        (* ***** Single Read SpecialFixcode ***** *)
        IF Head1.SaveRead AND NOT I_b_Head1SingleEnhanced AND I_b_Head1SpecialFixcode THEN
            Head_1_OutData[0] := 16#0A;
            Head_1_OutData[1] := 16#02;
            
            Head1.SglCommandActive := TRUE;
            Head1.EnhCommandActive := FALSE;
            Head1.Execute := TRUE;
            state_cmd1 := 1;
        END_IF;
        
        (* ***** Enhanced Read Words ***** *)
        IF Head1.SaveRead AND NOT I_b_Head1DataFixcode AND I_b_Head1SingleEnhanced AND NOT I_b_Head1SpecialFixcode THEN
            Head_1_OutData[0] := 16#19;
            Head_1_OutData[1] := WORD_TO_BYTE((INT_TO_WORD(SHL(I_i_Head1WordNum,  4)) OR 16#2));
            Head_1_OutData[2] := WORD_TO_BYTE(SHR(I_w_Head1WordAddress AND 16#FF00, 8));
            Head_1_OutData[3] := WORD_TO_BYTE(I_w_Head1WordAddress);
            
            Head1.EnhCommandActive := TRUE;
            Head1.Execute := TRUE;
            state_cmd1 := 1;
        END_IF;
        
        (* ***** Enhanced Read Fixcode ***** *)
        IF Head1.SaveRead AND I_b_Head1DataFixcode AND I_b_Head1SingleEnhanced AND NOT I_b_Head1SpecialFixcode THEN
            Head_1_OutData[0] := 16#1D;
            Head_1_OutData[1] := 16#02;
            
            Head1.EnhCommandActive := TRUE;
            Head1.Execute := TRUE;
            state_cmd1 := 1;
        END_IF;
        
        (* ***** Enhanced Read SpecialFixcode ***** *)
        IF Head1.SaveRead AND I_b_Head1SingleEnhanced AND I_b_Head1SpecialFixcode THEN
            Head_1_OutData[0] := 16#71;
            Head_1_OutData[1] := 16#02;
            
            Head1.EnhCommandActive := TRUE;
            Head1.Execute := TRUE;
            state_cmd1 := 1;
        END_IF;
        
        (* ***** Single Write Words ***** *)
        IF Head1.SaveWrite AND NOT I_b_Head1DataFixcode AND NOT I_b_Head1SingleEnhanced AND NOT I_b_Head1SpecialFixcode THEN
            Head_1_OutData[0] := 16#40;
            Head_1_OutData[1] := WORD_TO_BYTE((INT_TO_WORD(SHL(I_i_Head1WordNum, 4)) OR 16#2));
            Head_1_OutData[2] := WORD_TO_BYTE(SHR( I_w_Head1WordAddress AND 16#FF00,  8));
            Head_1_OutData[3] := WORD_TO_BYTE(I_w_Head1WordAddress);
            //Copy Write Data field to Out Data beginning at element [4]
            MEMCPY(srcAddr:=ADR(Head1Data.WriteData[0]) , destAddr:=ADR(Head_1_OutData[4]) , n:=SIZEOF(Head1Data.WriteData) );
			
            Head1.SglCommandActive := TRUE;
            Head1.EnhCommandActive := FALSE;
            Head1.Execute := TRUE;
            state_cmd1 := 1;
        END_IF;
        
        (* ***** Enhanced Write Words ***** *)
        IF Head1.SaveWrite AND NOT I_b_Head1DataFixcode AND I_b_Head1SingleEnhanced AND NOT I_b_Head1SpecialFixcode THEN
            Head_1_OutData[0] := 16#1A;
            Head_1_OutData[1] := WORD_TO_BYTE((INT_TO_WORD(SHL(I_i_Head1WordNum, 4)) OR 16#2));
            Head_1_OutData[2] := WORD_TO_BYTE(SHR( I_w_Head1WordAddress AND 16#FF00, 8));
            Head_1_OutData[3] := WORD_TO_BYTE(I_w_Head1WordAddress);
            //Copy Write Data field to Out Data beginning at element [4]		 
			MEMCPY(srcAddr:= ADR(Head1Data.WriteData[0]) , destAddr:=ADR(Head_1_OutData[4]) , n:=SIZEOF(Head1Data.WriteData) );		 
	 
            Head1.EnhCommandActive := TRUE;
            Head1.Execute := TRUE;
            state_cmd1 := 1;
        END_IF;
        
        (* ***** Single Write Fixcode ***** *) (* - default for IPC11, FixType = 11 & FixLen = 5 *)
        IF Head1.SaveWrite AND I_b_Head1DataFixcode AND NOT I_b_Head1SingleEnhanced AND NOT I_b_Head1SpecialFixcode THEN
            Head_1_OutData[0] := 16#1F;
            Head_1_OutData[1] := WORD_TO_BYTE((INT_TO_WORD(SHL(16#5,  4)) OR 16#2));
            Head_1_OutData[2] := 16#31; (* ASCII 11 = 0x3131, overwrite fixcode *)
            Head_1_OutData[3] := 16#31;
            //Copy Write Data field to Out Data beginning at element [4]
           MEMCPY(srcAddr:= ADR(Head1Data.WriteData[0]) , destAddr:=ADR(Head_1_OutData[4]) , n:=SIZEOF(Head1Data.WriteData) );
            	 
            Head1.SglCommandActive := TRUE;
            Head1.EnhCommandActive := FALSE;
            Head1.Execute := TRUE;
            state_cmd1 := 1;
        END_IF;
        
        (* ***** Single Write SpecialFixcode ***** *)
        IF Head1.SaveWrite AND NOT I_b_Head1SingleEnhanced AND I_b_Head1SpecialFixcode THEN
            Head_1_OutData[0] := 16#0D;
            Head_1_OutData[1] := WORD_TO_BYTE((INT_TO_WORD(SHL(I_i_Head1WordNum, 4)) OR 16#2));
            Head_1_OutData[2] := 16#0; (* reserved *)
            Head_1_OutData[3] := 16#0; (* reserved *)
            //Copy Write Data field to Out Data beginning at element [4]
            MEMCPY(srcAddr:= ADR(Head1Data.WriteData[0]) , destAddr:=ADR(Head_1_OutData[4]) , n:=SIZEOF(Head1Data.WriteData ));
		 
            Head1.SglCommandActive := TRUE;
            Head1.EnhCommandActive := FALSE;
            Head1.Execute := TRUE;
            state_cmd1 := 1;
        END_IF;
        
        (* ***** Special Command ***** *)
        IF Head1.SaveSpecialCommand AND NOT I_b_Head1SpecialFixcode THEN
        (* Copy SpecialCommand-Array into Output-Array *)
            //Copy the whole SpecialCommand data field to the Output Data
			 MEMCPY(srcAddr:=ADR(Head1Data.SpecialCommand[0]) , destAddr:=ADR(Head_1_OutData[0]) , n:=SIZEOF(Head1Data.SpecialCommand) );		 
			
            Head1.SglCommandActive := TRUE;
            Head1.EnhCommandActive := FALSE;
            Head1.Execute := TRUE;
            state_cmd1 := 1;
        END_IF;
    END_IF;
    
(* ***** Handle communication and analysis for channel 1 ***** *)
    CASE state_cmd1 OF
            
        0:  (* ***** Idle state ***** *)
//        IF NOT I_b_Head1SingleEnhanced
//			AND NOT	I_b_Head1DataFixcode
//			AND NOT	I_b_Head1SpecialFixcode
//			AND NOT	I_b_Head1SpecialCommand
//			AND NOT	I_b_Head1Read
//			AND NOT	I_b_Head1Write
//			AND NOT	I_b_Head1Quit
//			THEN
			O_b_Head1Done := FALSE;
			//O_b_Head1NoDataCarrier := FALSE;
//		END_IF

        1:  (* ***** Execution ***** *)
            IF Head1.Execute AND NOT Head1.TransfToHead THEN
                
                Head1.Busy := TRUE;
                O_b_Head1Busy := TRUE;
                Head1.Done := FALSE;
                O_b_Head1Done := FALSE;
                Head1.Error := FALSE;
                O_b_Head1Error := FALSE;
                Head1.SendOK := FALSE;
                Head1.ReceiveOK := FALSE;
                Head1.NoDataCarrier := FALSE;
                O_b_Head1NoDataCarrier := FALSE;
                Head1.NewData := FALSE;
                Head1.TimeoutActive := TRUE;
                Head1.TimeoutOccurred := FALSE;
                Head1.TransfToHead := TRUE;
                Head1.SaveRead := FALSE;
                Head1.SaveWrite := FALSE;
                Head1.SaveQuit := FALSE;
                Head1.SaveSpecialCommand := FALSE;
                
                (* Invert togglebit => new telegram is available *)
                IF Memory.Togglebit <> 1 THEN
                    Head_1_OutData[1] := Head_1_OutData[1] OR 16#1;
                ELSE
                    Head_1_OutData[1] := Head_1_OutData[1] AND 16#FE;
                END_IF;
                
               		HwOut:= Head_1_OutData ; (* Write on BUS *)
               
                 
                    state_cmd1 := state_cmd1 + 1; (* Go to next state *)
                
            END_IF;
            
            
        2:(* ***** Analyze InData ***** *)
        (* Receive Telegram *)
            IF Head1.NewData THEN
                
                Head1.NewData := FALSE;
                (* Transfer status & reply counter to output *)
                O_B_Head1Status := Head_1_InData[2];
                O_B_Head1ReplyCounter := Head_1_InData[3];
                
                (* Analyze status *)
                IF Head_1_InData[2] = 16#FF THEN
                    Head1.SendOK := TRUE;
                    Head1.TransfToHead := FALSE;
                ELSE
                    Head1.Execute := FALSE;
                    Head1.ReceiveOK := TRUE;
                    Head1.SglCommandActive := FALSE;
                    Head1.TimeoutActive := FALSE;
                    Head1.Busy := FALSE;
                    O_b_Head1Busy := FALSE;
                    Head1.Done := TRUE;
                    O_b_Head1Done := TRUE;
                    state_cmd1 := 0; (* Go to idle state *)
                END_IF;
                
                IF Head_1_InData[2] = 16#0 THEN
                    Head1.NoDataCarrier := FALSE;
                    O_b_Head1NoDataCarrier := FALSE;
                    Head1.Error := FALSE;      //new in 3.0
                    O_b_Head1Error := FALSE;       //new in 3.0
                END_IF;
                
                IF Head_1_InData[2] = 16#5 THEN
                    Head1.NoDataCarrier := TRUE;
                    O_b_Head1NoDataCarrier := TRUE;
                    Head1.Error := FALSE;      //new in 3.0
                    O_b_Head1Error := FALSE;       //new in 3.0
                END_IF;
                
                (* Error states *)
                IF Head_1_InData[2] = 16#4
                    OR Head_1_InData[2] = 16#6
                    OR Head_1_InData[2] = 16#7
                    OR Head_1_InData[2] = 16#9
                    OR Head_1_InData[2] = 16#A
                    OR Head_1_InData[2] = 16#E THEN
                    Head1.Error := TRUE;
                    O_b_Head1Error := TRUE;
                END_IF;
                
                (* Different output behaviour during active enhanced command *)
                IF Head1.EnhCommandActive THEN
                    state_cmd1 := 2; (* Receive new telegram *)
                    Head1.Busy := TRUE;
                    O_b_Head1Busy := TRUE;
                    IF Head_1_InData[2] = 16#0 THEN
                        Head1.Done := TRUE;
                        O_b_Head1Done := TRUE;
                    ELSE
                        Head1.Done := FALSE;
                        O_b_Head1Done := FALSE;
                    END_IF;
                END_IF;
            END_IF;
    END_CASE;
	
	
END_IF;

(* ***** Watchdog ***** *)
//Watchdog1(IN := Head1.TimeoutActive,PT := I_T_Timeout);

IF (Watchdog1.Q AND temp) THEN
    Head1.TimeoutActive := FALSE;
    Head1.TimeoutOccurred := TRUE;
    Head1.SendOK := FALSE;
    Head1.ReceiveOK := FALSE;
    Head1.SglCommandActive := FALSE;
    Head1.EnhCommandActive := FALSE;
    Head1.Execute := FALSE;
    Head1.TransfToHead := FALSE;
    Head1.Error := TRUE;
    O_b_Head1Error := TRUE;
    Head1.Busy := FALSE;
    O_b_Head1Busy := FALSE;
    Head1.Done := TRUE;
    O_b_Head1Done := TRUE;
END_IF

END_FUNCTION_BLOCK

// ---- POUs/Programs/OP10/OP10_MAIN.TcPOU
PROGRAM OP10_MAIN
VAR

	OP10A_ROBO_MANUL_TRG: R_TRIG;
	OP10A_ROBO_AUTO_TRG	: R_TRIG;
	Bowl_A_ON_Timer		: TON;
	Bowl_A_OFF_Timer	: TON;
	Bowl_B_ON_Timer		: TON;
	Bowl_B_OFF_Timer	: TON;
	OP10A_ROBO_ERR		: TON;
	OP10B_ROBO_ERR		: TON;
	SRV_HOME			: BOOL;	
	OP10_ROBO			: INT;
	OP10A_ROBO_MANUAL	: INT;
	OP10A_ROBO_AUTO		: INT;
	// TEMP
	TEMP_40				: BOOL;

	

	
	OP10B_ROBO_MANUL_TRG: R_TRIG;
	OP10B_ROBO_AUTO_TRG: R_TRIG;
	OP10B_ROBO_MANUAL: INT;
	OP10B_ROBO_AUTO: INT;
END_VAR

VAR PERSISTENT
	OP10A_ROBO_ERR_TIME	: TIME;
	OP10B_ROBO_ERR_TIME	: TIME;
END_VAR

OP10_MANUAL();
OP10_SERVO();
OP10_HOMING();
OP10A_AUTO();
OP10B_AUTO();
//OP10_AUTO();
Bowl_Control();
OP10A_Camera_FB();
OP10B_Camera_FB();
OP10A_OP10B_DRUM_FEEDER();
OP10B_Conveyor_Prog();
OP10A_Conveyor_Prog();
//OP10_Body_Camera_Seq();
Body_Singulation_Seq();

OP10A_MODE_BLOCK(
	ModeWord:= OP10A_MODE_WORD, 
	HomeConditionOK:= OP10A_ALL_HOME,//OP10A_ALL_HOME, 
	OperationEnable:= OperationEnable, 
	StartPB:= OP10A_STRT_PB, 
	SafetyAndNOError:= NOT OP10A_ERR,//(NOT OP10A_ERR), 
	ModeAck:= 1, 
	HomingINProgress:= , 
	TempHomeOK:=  , 
	ResetPB:= Servo_Reset, 
	AutoSelected=> OP10A_AUTO_SELECTED, 
	ManualSelected=> OP10A_MANUAL_SELECTED, 
	StepSelected=> OP10A_STEP_SELECTED, 
	ModeSelAck_Indication=> , 
	StatusDisplay=> , 
	AutoRunning:=OP10A_AUTO_RUNNING, 
	StepRunning:=OP10A_STEP_RUNNING , 
	StartEnable:=OP10A_START_ENABLE , 
	MachineStop:=OP10A_MACHINE_STOP );
	
	
	OP10A_ROBO_MANUL_TRG(CLK:=OP10A_MANUAL_SELECTED , Q=> );
	OP10A_ROBO_AUTO_TRG(CLK:=NOT OP10A_MANUAL_SELECTED , Q=> );
	
IF OP10A_ROBO_MANUL_TRG.Q THEN
	OP10A_ROBO_MANUAL	:= 1;
END_IF

IF OP10A_ROBO_AUTO_TRG.Q THEN
	OP10A_ROBO_AUTO		:= 1;
END_IF


CASE OP10A_ROBO_MANUAL OF 
	1: OP10A_ROBO_PRGM_RST				:= TRUE;
		OP10A_ROBO_MANUAL				:= 5;
		
	5: IF (OP10A_ROBO_PRGM_RST =TRUE) AND (NOT OP10A_Program_Execute) THEN
		OP10A_ROBO_PRGM_RST				:= FALSE;
		O10A_ROB_MAN_AUTO_MODE_Q709_2	:= FALSE;
		OP10A_ROBO_MANUAL				:= 10;
		END_IF
END_CASE

CASE OP10A_ROBO_AUTO OF 
	1: OP10A_ROBO_PRGM_RST				:= TRUE;
		OP10A_ROBO_AUTO					:= 5;

	5: IF (OP10A_ROBO_PRGM_RST =TRUE) AND (NOT OP10A_Program_Execute) THEN
		OP10A_ROBO_PRGM_RST				:= FALSE;
		O10A_ROB_MAN_AUTO_MODE_Q709_2	:= TRUE;
		OP10A_ROBO_AUTO					:= 10;
		END_IF
END_CASE


OP10A_ROBO_ERR(IN:=	NOT(OP10A_Auto_Operation_Enable AND OP10A_Mirror_Auto_enable AND OP10A_Servo_ON_OFF_Status) , PT:=OP10A_ROBO_ERR_TIME, Q=> , ET=> );
			
IF (OP10A_AUTO_SELECTED AND NOT OP10A_ROBO_PRGM_RST AND OP10A_ROBO_ERR.Q) OR OP10A_H_Error OR OP10A_L_Error OR 
		OP10_SRV_FRST_PCKBDY_CNT.Axis_Error OR OP10_SRV_SCND_PCKBDY_CNT.Axis_Error OR(OP10A_CYLINDER_ERR<>0) OR 
			(OP10A_SRV_LH_BDYANG_CNT.Axis_Error AND NOT OP10A_BDY1_PCK_BYPAS) OR (OP10A_SRV_RH_BDYANG_CNT.Axis_Error AND 
				NOT OP10A_BDY2_PCK_BYPAS) OR (OP10A_SRV_LH_BDYGRP_CNT.Axis_Error  AND NOT OP10A_BDY1_PCK_BYPAS) OR 
					(OP10A_SRV_RH_BDYGRP_CNT.Axis_Error AND NOT OP10A_BDY2_PCK_BYPAS)  THEN
//OP10A_ERR		:= TRUE;
ELSE
OP10A_ERR		:= FALSE;	
END_IF

IF SRV_HOME	THEN
IF OP10A_Rbt_In_Home AND OP10B_Rbt_In_Home THEN
OP10_A_SRV_FST_BDYPCK_HME	:=1;
OP10_A_SRV_SCND_BDYPCK_HME	:=1;	
END_IF
OP10A_A_SRV_LH_GRPHME       :=1;
OP10A_A_SRV_RH_GRPHME       :=1;
OP10A_SRV_LH_BDYANG_HME     :=1;
OP10A_SRV_RH_BDYANG_HME     :=1;
IF OP10A_ALL_HOME THEN
OP10_A_SRV_FST_BDYPCK_HME	:=0;
OP10_A_SRV_SCND_BDYPCK_HME	:=0;
OP10A_A_SRV_LH_GRPHME       :=0;
OP10A_A_SRV_RH_GRPHME       :=0;
OP10A_SRV_LH_BDYANG_HME     :=0;
OP10A_SRV_RH_BDYANG_HME     :=0;	
SRV_HOME					:=0;
END_IF	
END_IF
(*
O10A_BDY_LNR1_AIR_PURGE_Q101_3:=I10A_BDY_BWL_RUN_I101_3;
O10A_BDY_LNR2_AIR_PURGE_Q101_4:=I10A_BDY_BWL_RUN_I101_3;
O10B_BDY_LNR1_AIR_PURGE_Q201_3:=I10B_BDY_BWL_RUN_I201_3;
O10B_BDY_LNR2_AIR_PURGE_Q201_4:=I10B_BDY_BWL_RUN_I201_3;

O10A_HPR_MTR_FWD_Q100_0			:=I10A_HPR_OFF_ON_I100_4;
O10A_HPR_TWR_LMP_GREEN_Q100_6	:=I10A_HPR_OFF_ON_I100_4;
//O10A_BDY_BOWL_ON_Q101_0			:=I10A_BDY_BOWL_OFF_ON_I100_5;
O10A_BDY_LNR_FEED1_ON_Q101_1	:=I10A_BDY_LNR1_OFF_ON_I100_6 OR I10A_BDY_LNR2_OFF_ON_I100_7;
O10A_BDY_LNR_FEED2_ON_Q101_2    :=I10A_BDY_LNR1_OFF_ON_I100_6 OR I10A_BDY_LNR2_OFF_ON_I100_7;

O10B_HPR_MTR_FWD_Q200_0		   := I10B_HPR_OFF_ON_I200_4;
O10B_HPR_TWR_LMP_GREEN_Q200_6  := I10B_HPR_OFF_ON_I200_4;
//O10B_BDY_BOWL_ON_Q201_0        := I10B_BDY_BOWL_OFF_ON_I200_5;
O10B_BDY_LNR_FEED1_ON_Q201_1   := I10B_BDY_LNR1_OFF_ON_I200_6 OR I10B_BDY_LNR2_OFF_ON_I200_7;
O10B_BDY_LNR_FEED2_ON_Q201_2   := I10B_BDY_LNR1_OFF_ON_I200_6 OR I10B_BDY_LNR2_OFF_ON_I200_7;


Bowl_A_ON_Timer(IN:= NOT I10A_BDY_LNR_FEED2_OVRFLW_I101_7,PT:=T#2S);
Bowl_A_OFF_Timer(IN:= I10A_BDY_LNR_FEED1_OVRFLW_I101_6,PT:=T#2S);

Bowl_B_ON_Timer(IN:= NOT I10B_BDY_LNR_FEED2_OVRFLW_I201_7,PT:=T#2S);
Bowl_B_OFF_Timer(IN:=I10B_BDY_LNR_FEED1_OVRFLW_I201_6,PT:=T#2S);

IF I10A_BDY_BOWL_OFF_ON_I100_5 THEN
	IF 	Bowl_A_OFF_Timer.Q THEN
		O10A_BDY_BOWL_ON_Q101_0:=1;
	END_IF
	IF Bowl_A_ON_Timer.Q THEN
		O10A_BDY_BOWL_ON_Q101_0:=0;
	END_IF
ELSE
	O10A_BDY_BOWL_ON_Q101_0:=1;
END_IF

IF I10B_BDY_BOWL_OFF_ON_I200_5 THEN
	IF 	Bowl_B_OFF_Timer.Q THEN
		O10B_BDY_BOWL_ON_Q201_0:=1;
	END_IF
	IF Bowl_B_ON_Timer.Q THEN
		O10B_BDY_BOWL_ON_Q201_0:=0;
	END_IF
ELSE
	O10B_BDY_BOWL_ON_Q201_0:=1;	
END_IF	*)

	OP10B_MODE_BLOCK(
	ModeWord:= OP10B_MODE_WORD, 
	HomeConditionOK:= 1,//OP10B_ALL_HOME,
	OperationEnable:= OperationEnable, 
	StartPB:= OP10B_STRT_PB, 
	SafetyAndNOError:= NOT OP10B_ERR, 
	ModeAck:= 1, 
	HomingINProgress:= , 
	TempHomeOK:=  , 
	ResetPB:= Servo_Reset, 
	AutoSelected=> OP10B_AUTO_SELECTED, 
	ManualSelected=> OP10B_MANUAL_SELECTED, 
	StepSelected=> OP10B_STEP_SELECTED, 
	ModeSelAck_Indication=> , 
	StatusDisplay=> , 
	AutoRunning:=OP10B_AUTO_RUNNING, 
	StepRunning:=OP10B_STEP_RUNNING , 
	StartEnable:=OP10B_START_ENABLE , 
	MachineStop:=OP10B_MACHINE_STOP ); 

////////////////

OP10B_ROBO_MANUL_TRG(CLK:=OP10B_MANUAL_SELECTED , Q=> );
	OP10B_ROBO_AUTO_TRG(CLK:=NOT OP10B_MANUAL_SELECTED , Q=> );
	
IF OP10B_ROBO_MANUL_TRG.Q THEN
	OP10B_ROBO_MANUAL	:= 1;
END_IF

IF OP10B_ROBO_AUTO_TRG.Q THEN
	OP10B_ROBO_AUTO		:= 1;
END_IF


CASE OP10B_ROBO_MANUAL OF 
	1: OP10B_ROBO_PRGM_RST				:= TRUE;
		OP10B_ROBO_MANUAL				:= 5;
		
	5: IF (OP10B_ROBO_PRGM_RST =TRUE) AND (NOT OP10B_Program_Execute) THEN
		OP10B_ROBO_PRGM_RST				:= FALSE;
		O10B_ROB_MAN_AUTO_MODE_Q709_3	:= FALSE;
		OP10B_ROBO_MANUAL				:= 10;
		END_IF
END_CASE

CASE OP10B_ROBO_AUTO OF 
	1: OP10B_ROBO_PRGM_RST				:= TRUE;
		OP10B_ROBO_AUTO					:= 5;

	5: IF (OP10B_ROBO_PRGM_RST =TRUE) AND (NOT OP10B_Program_Execute) THEN
		OP10B_ROBO_PRGM_RST				:= FALSE;
		O10B_ROB_MAN_AUTO_MODE_Q709_3	:= TRUE;
		OP10B_ROBO_AUTO					:= 10;
		END_IF
END_CASE


//#####################		OP10B_ERROR		########################

OP10B_ROBO_ERR(IN:= NOT(OP10B_Auto_Operation_Enable AND OP10B_Mirror_Auto_enable AND OP10B_Servo_ON_OFF_Status), PT:=OP10B_ROBO_ERR_TIME, Q=> , ET=> );	

IF (OP10B_AUTO_SELECTED AND NOT OP10B_ROBO_PRGM_RST AND OP10B_ROBO_ERR.Q) OR OP10B_H_Error OR OP10B_L_Error OR 
		OP10_SRV_FRST_PCKBDY_CNT.Axis_Error OR OP10_SRV_SCND_PCKBDY_CNT.Axis_Error OR (OP10B_CYLINDER_ERR<>0) OR 
			(OP10B_SRV_LH_BDYANG_CNT.Axis_Error AND NOT OP10B_BDY1_PCK_BYPAS) OR (OP10B_SRV_RH_BDYANG_CNT.Axis_Error AND 
				NOT OP10B_BDY2_PCK_BYPAS) OR (OP10B_SRV_LH_BDYGRP_CNT.Axis_Error AND NOT OP10B_BDY1_PCK_BYPAS) OR 
				(OP10B_SRV_RH_BDYGRP_CNT.Axis_Error AND NOT OP10B_BDY2_PCK_BYPAS)THEN 
OP10B_ERR		:= TRUE;
ELSE
OP10B_ERR		:= FALSE;	
END_IF

END_PROGRAM

// ---- POUs/Programs/OP10/OP10_MANUAL.TcPOU
PROGRAM OP10_MANUAL
VAR
//OP10A
	OP10A_O_HORZ_MANUALPB1							: BOOL;
	OP10A_O_HORZ_MANUALPB2							: BOOL;
	OP10A_O_VERT_MANUALPB1							: BOOL;
	OP10A_O_VERT_MANUALPB2							: BOOL;
	OP10A_M_O_LHGRIP_ONOFF							: BOOL;
	OP10A_M_O_RHGRIP_ONOFF							: BOOL;
	OP10A_M_O_LHPUSH_CYL							: BOOL;
	OP10A_M_O_RHPUSH_CYL							: BOOL;	
	OP10A_O_0DEGRE_MANUALPB1						: BOOL;
	OP10A_O_180DEGRE_MANUALPB2						: BOOL;
	OP10A_M_LNR1_ONOFF								: BOOL;
	OP10A_M_LNR2_ONOFF								: BOOL;
	OP10A_M_BOWL_ONOFF								: BOOL;
	OP10A_M_HOPPER_ONOFF							: BOOL;
	OP10A_M_LH_REJ_WRK								: BOOL;
	OP10A_M_LH_REJ_HOME								: BOOL;
	OP10A_M_RH_REJ_HOME								: BOOL;
	OP10A_M_RH_REJ_WRK								: BOOL;
	OP10_FRT_BDY_SING_HME							: BOOL;
	OP10_FRT_BDY_SING_WRK							: BOOL;	
	OP10_SEC_BDY_SING_HME							: BOOL;
	OP10_SEC_BDY_SING_WRK							: BOOL;	
	
	
//OP10B                                     		
	OP10B_O_HORZ_MANUALPB1							: BOOL;
	OP10B_O_HORZ_MANUALPB2							: BOOL;
	OP10B_O_VERT_MANUALPB1							: BOOL;
	OP10B_O_VERT_MANUALPB2							: BOOL;
	OP10B_M_O_LHGRIP_ONOFF							: BOOL;
	OP10B_M_O_RHGRIP_ONOFF							: BOOL;
	OP10B_M_O_LHPUSH_CYL							: BOOL;
	OP10B_M_O_RHPUSH_CYL							: BOOL;
	OP10B_O_0DEGRE_MANUALPB1						: BOOL;
	OP10B_O_180DEGRE_MANUALPB2						: BOOL;
	OP10B_M_LNR1_ONOFF								: BOOL;
	OP10B_M_LNR2_ONOFF								: BOOL;
	OP10B_M_BOWL_ONOFF								: BOOL;
	OP10B_M_HOPPER_ONOFF							: BOOL;
	OP10B_M_LH_REJ_HOME								: BOOL;
	OP10B_M_LH_REJ_WRK								: BOOL;
	OP10B_M_RH_REJ_HOME								: BOOL;
	OP10B_M_RH_REJ_WRK								: BOOL;
	
// ALARM BITS

	OP10A_HORZ_CYL_A1								: BOOL;
	OP10A_HORZ_CYL_A2								: BOOL;
	OP10A_HORZ_CYL_A3								: BOOL;
	OP10A_HORZ_CYL_A4								: BOOL;
	OP10A_HORZ_CYL_A5								: BOOL;
	OP10A_VERT_CYL_A1								: BOOL;
	OP10A_VERT_CYL_A2								: BOOL;
	OP10A_VERT_CYL_A3								: BOOL;
	OP10A_VERT_CYL_A4								: BOOL;
	OP10A_VERT_CYL_A5								: BOOL;
	OP10A_DEGREE_CYL_A1								: BOOL;
	OP10A_DEGREE_CYL_A2								: BOOL;
	OP10A_DEGREE_CYL_A3								: BOOL;
	OP10A_DEGREE_CYL_A4								: BOOL;
	OP10A_DEGREE_CYL_A5								: BOOL;
	OP10A_LH_GRP_A1									: BOOL;
	OP10A_LH_GRP_A2									: BOOL;
	OP10A_LH_GRP_A3									: BOOL;
	OP10A_LH_GRP_A4									: BOOL;
	OP10A_LH_GRP_A5									: BOOL;
	OP10A_RH_GRP_A1									: BOOL;
	OP10A_RH_GRP_A2									: BOOL;
	OP10A_RH_GRP_A3									: BOOL;
	OP10A_RH_GRP_A4									: BOOL;
	OP10A_RH_GRP_A5									: BOOL;
	OP10A_LH_PUSH_A1								: BOOL;
	OP10A_LH_PUSH_A2								: BOOL;
	OP10A_LH_PUSH_A3								: BOOL;
	OP10A_LH_PUSH_A4								: BOOL;
	OP10A_LH_PUSH_A5								: BOOL;
	OP10A_RH_PUSH_A1								: BOOL;
	OP10A_RH_PUSH_A2								: BOOL;
	OP10A_RH_PUSH_A3								: BOOL;
	OP10A_RH_PUSH_A4								: BOOL;
	OP10A_RH_PUSH_A5								: BOOL;
	OP10A_LH_REJ_A1									: BOOL;
	OP10A_LH_REJ_A2									: BOOL;
	OP10A_LH_REJ_A3									: BOOL;
	OP10A_LH_REJ_A4									: BOOL;
	OP10A_LH_REJ_A5									: BOOL;
	OP10A_RH_REJ_A1									: BOOL;
	OP10A_RH_REJ_A2									: BOOL;
	OP10A_RH_REJ_A3									: BOOL;
	OP10A_RH_REJ_A4									: BOOL;
	OP10A_RH_REJ_A5									: BOOL;
	OP10B_HORZ_CYL_A1								: BOOL;
	OP10B_HORZ_CYL_A2								: BOOL;
	OP10B_HORZ_CYL_A3								: BOOL;
	OP10B_HORZ_CYL_A4								: BOOL;
	OP10B_HORZ_CYL_A5								: BOOL;
	OP10B_VERT_CYL_A1								: BOOL;
	OP10B_VERT_CYL_A2								: BOOL;
	OP10B_VERT_CYL_A3								: BOOL;
	OP10B_VERT_CYL_A4								: BOOL;
	OP10B_VERT_CYL_A5								: BOOL;
	OP10B_DEGREE_CYL_A1								: BOOL;
	OP10B_DEGREE_CYL_A2								: BOOL;
	OP10B_DEGREE_CYL_A3								: BOOL;
	OP10B_DEGREE_CYL_A4								: BOOL;
	OP10B_DEGREE_CYL_A5								: BOOL;
	OP10B_LH_GRP_A1									: BOOL;
	OP10B_LH_GRP_A2									: BOOL;
	OP10B_LH_GRP_A3									: BOOL;
	OP10B_LH_GRP_A4									: BOOL;
	OP10B_LH_GRP_A5									: BOOL;
	OP10B_RH_GRP_A1									: BOOL;
	OP10B_RH_GRP_A2									: BOOL;
	OP10B_RH_GRP_A3									: BOOL;
	OP10B_RH_GRP_A4									: BOOL;
	OP10B_RH_GRP_A5									: BOOL;
	OP10B_LH_PUSH_A1								: BOOL;
	OP10B_LH_PUSH_A2								: BOOL;
	OP10B_LH_PUSH_A3								: BOOL;
	OP10B_LH_PUSH_A4								: BOOL;
	OP10B_LH_PUSH_A5								: BOOL;
	OP10B_RH_PUSH_A1								: BOOL;
	OP10B_RH_PUSH_A2								: BOOL;
	OP10B_RH_PUSH_A3								: BOOL;
	OP10B_RH_PUSH_A4								: BOOL;
	OP10B_RH_PUSH_A5								: BOOL;
	OP10B_LH_REJ_A1									: BOOL;
	OP10B_LH_REJ_A2									: BOOL;
	OP10B_LH_REJ_A3									: BOOL;
	OP10B_LH_REJ_A4									: BOOL;
	OP10B_LH_REJ_A5									: BOOL;
	OP10B_RH_REJ_A1									: BOOL;
	OP10B_RH_REJ_A2									: BOOL;
	OP10B_RH_REJ_A3									: BOOL;
	OP10B_RH_REJ_A4									: BOOL;
	OP10B_RH_REJ_A5									: BOOL;	
	OP10_BDY_SING_FRT_A1							: BOOL;
	OP10_BDY_SING_FRT_A2							: BOOL;
	OP10_BDY_SING_FRT_A3							: BOOL;
	OP10_BDY_SING_FRT_A4							: BOOL;
	OP10_BDY_SING_FRT_A5							: BOOL;	
	OP10_BDY_SING_SEC_A1							: BOOL;
	OP10_BDY_SING_SEC_A2							: BOOL;
	OP10_BDY_SING_SEC_A3							: BOOL;
	OP10_BDY_SING_SEC_A4							: BOOL;
	OP10_BDY_SING_SEC_A5							: BOOL;	
	
	
	

//INT

	OP10A_HORZ_CYL_STUS								: INT;
	OP10A_VERT_CYL_STUS								: INT;
	OP10A_DEGREE_CYL_STUS							: INT;
	OP10A_LH_GRP_STATS								: INT;
	OP10A_RH_GRP_STUS								: INT;
	OP10A_LH_PUSH_STUS								: INT;
	OP10A_RH_PUSH_STUS								: INT;
	OP10B_HORZ_CYL_STUS								: INT;
	OP10B_VERT_CYL_STUS								: INT;
	OP10B_DEGREE_CYL_STUS							: INT;
	OP10B_LH_GRP_STATS								: INT;
	OP10B_RH_GRP_STUS								: INT;
	OP10B_LH_PUSH_STUS								: INT;
	OP10B_RH_PUSH_STUS								: INT;
                              				
// BOOL                             				
	OP10A_H_LNR1_ONOFF								: BOOL;
	OP10A_H_LNR2_ONOFF								: BOOL;
	OP10A_H_BOWL_ONOFF								: BOOL;
	OP10A_H_HOPPER_ONOFF							: BOOL;
	OP10B_H_LNR1_ONOFF								: BOOL;
	OP10B_H_LNR2_ONOFF								: BOOL;
	OP10B_H_BOWL_ONOFF								: BOOL;
	OP10B_H_HOPPER_ONOFF							: BOOL;

	
	
	
HMI_TRIAL_SWITH_GOKUL_2							:BOOL;	
	
TEMP	: BOOL;
	temp1: BOOL;
	temp2: BOOL;
	OP10_BDY_SING_FRT_STATUS: INT;
	OP10_BDY_SING_SEC_STATUS: INT;




	OP10B_PARLLEL: INT;
	OP10A_PARALLEL: INT;
END_VAR

VAR RETAIN

END_VAR

//#############################		OP10A		###############################

IF OP10A_MANUAL_SELECTED THEN

//OP10A
	OP10A_M_LNR1_ONOFF							:= OP10A_H_LNR1_ONOFF;
	OP10A_M_LNR2_ONOFF          				:= OP10A_H_LNR2_ONOFF;
	OP10A_M_BOWL_ONOFF          				:= OP10A_H_BOWL_ONOFF;
	OP10A_M_HOPPER_ONOFF        				:= OP10A_H_HOPPER_ONOFF;	

CASE OP10_CYL_NO OF                 		
	                                		
	1: IF OP10_HOME THEN            		
		OP10A_O_HORZ_MANUALPB1					:=TRUE;
		OP10A_O_HORZ_MANUALPB2					:=FALSE;
		END_IF                      			
		IF OP10_WORK THEN           			
		OP10A_O_HORZ_MANUALPB1					:=FALSE;
		OP10A_O_HORZ_MANUALPB2					:=TRUE;
		END_IF                      			
                                    			
	2: IF OP10_HOME THEN            			
		OP10A_O_VERT_MANUALPB1					:=TRUE;
		OP10A_O_VERT_MANUALPB2					:=FALSE;
		END_IF                      		
		IF OP10_WORK THEN           		
		OP10A_O_VERT_MANUALPB1					:=FALSE;
		OP10A_O_VERT_MANUALPB2					:=TRUE;
		END_IF                      			
		                            			
	4:IF OP10_HOME THEN             			
		OP10A_O_0DEGRE_MANUALPB1				:=TRUE;
		OP10A_O_180DEGRE_MANUALPB2				:=FALSE;
		END_IF                      			
		IF OP10_WORK THEN           			
		OP10A_O_0DEGRE_MANUALPB1				:=FALSE;
		OP10A_O_180DEGRE_MANUALPB2				:=TRUE;
		END_IF                      		
                            		
	9: IF OP10_HOME THEN            		
		OP10A_M_LH_REJ_HOME						:=TRUE;
		OP10A_M_LH_REJ_WRK		 				:=FALSE;
		END_IF                      			
		IF OP10_WORK THEN           			
		OP10A_M_LH_REJ_HOME						:=FALSE;
		OP10A_M_LH_REJ_WRK	 					:=TRUE;
		END_IF                      			
		                            			
	10: IF OP10_HOME THEN           			
		OP10A_M_RH_REJ_HOME						:=TRUE;
		OP10A_M_RH_REJ_WRK	 	 				:=FALSE;
		END_IF                      			
		IF OP10_WORK THEN           			
		OP10A_M_RH_REJ_HOME						:=FALSE;
		OP10A_M_RH_REJ_WRK	 					:=TRUE;
		END_IF	                    		
		                            		                     		
		                            		
	13: IF OP10_HOME THEN           		
		OP10A_M_O_LHGRIP_ONOFF					:=FALSE;
		END_IF                      			
		IF OP10_WORK THEN           			
		OP10A_M_O_LHGRIP_ONOFF					:=TRUE;
		END_IF                      			
		                            			
	14:	IF OP10_HOME THEN           			
		OP10A_M_O_RHGRIP_ONOFF					:=FALSE;
		END_IF                      			
		IF OP10_WORK THEN           	    	
		OP10A_M_O_RHGRIP_ONOFF					:=TRUE;
		END_IF                      			
		                            			
	15: IF OP10_HOME THEN           			
		OP10A_M_O_LHPUSH_CYL					:=FALSE;
		END_IF                      		
		IF OP10_WORK THEN           		
		OP10A_M_O_LHPUSH_CYL					:=TRUE;
		END_IF                      			
		                            			
	16: IF OP10_HOME THEN           			
		OP10A_M_O_RHPUSH_CYL					:=FALSE;
		END_IF                      			
		IF OP10_WORK THEN           			
		OP10A_M_O_RHPUSH_CYL					:=TRUE;
		END_IF                              	
		                                    	
	17: IF OP10_HOME THEN           			
		OP10_FRT_BDY_SING_HME					:=TRUE;
		OP10_FRT_BDY_SING_WRK 	 				:=FALSE;
		END_IF                      		
		IF OP10_WORK THEN           		
		OP10_FRT_BDY_SING_HME	 				:=FALSE;
		OP10_FRT_BDY_SING_WRK 					:=TRUE;
		END_IF                              	
                                            	
	18: IF OP10_HOME THEN           			
		OP10_SEC_BDY_SING_HME					:=TRUE;
		OP10_SEC_BDY_SING_WRK		 			:=FALSE;
		END_IF                      		
		IF OP10_WORK THEN           		
		OP10_SEC_BDY_SING_HME					:=FALSE;
		OP10_SEC_BDY_SING_WRK					:=TRUE;
		END_IF                              	
                    		                	
		                            	    	
END_CASE

CASE OP10_SERVO_NO OF               	
	                                	
	1: OP10A_SRV_O_CNVY_STUS.jogPos				:= OP10_JOG_POSITIVE AND NOT OP10_JOG_NEGATIVE;
	   OP10A_SRV_O_CNVY_STUS.jogNeg				:= OP10_JOG_NEGATIVE AND NOT OP10_JOG_POSITIVE;
	   OP10A_SRV_O_CNVY_CNT.Bsethome	        := OP10A_SET_HOME;
	   OP10A_SRV_O_CNVY_STUS.targetPositon	    := OP10A_TARGET_POSITION;
	   OP10A_SRV_O_CNVY_STUS.moveAbsolute	    := OP10A_MOVE_TARGET;
	   OP10A_SRV_ACT_POS						:= OP10A_SRV_O_CNVY_STUS.actualPosition;
	   OP10A_SRV_FAULT							:= OP10A_CONVEYOR.bAxisError;
	   OP10A_SRV_ENABLE							:= OP10A_CONVEYOR.bAxisEnabled;

	    
	3: OP10A_SRV_LH_BDYGRP_STUS.jogPos			:= OP10_JOG_POSITIVE AND NOT OP10_JOG_NEGATIVE;
	   OP10A_SRV_LH_BDYGRP_STUS.jogNeg      	:= OP10_JOG_NEGATIVE AND NOT OP10_JOG_POSITIVE;  
	   OP10A_SRV_LH_BDYGRP_CNT.Axis_Home_Cmd	:= OP10A_SET_HOME;
	   OP10A_SRV_LH_BDYGRP_STUS.targetPositon	:= OP10A_TARGET_POSITION;
	   OP10A_SRV_LH_BDYGRP_STUS.moveAbsolute	:= OP10A_MOVE_TARGET;
	   OP10A_SRV_ACT_POS						:= OP10A_SRV_LH_BDYGRP_STUS.actualPosition;
	   OP10A_SRV_FAULT							:= OP10A_LH_GRIPR.bAxisError;
	   OP10A_SRV_ENABLE							:= OP10A_LH_GRIPR.bAxisEnabled;
	   
	4: OP10A_SRV_RH_BDYGRP_STUS.jogPos			:= OP10_JOG_POSITIVE AND NOT OP10_JOG_NEGATIVE;
	   OP10A_SRV_RH_BDYGRP_STUS.jogNeg   		:= OP10_JOG_NEGATIVE AND NOT OP10_JOG_POSITIVE;
	   OP10A_SRV_RH_BDYGRP_CNT.Axis_Home_Cmd	:= OP10A_SET_HOME;
	   OP10A_SRV_RH_BDYGRP_STUS.targetPositon	:= OP10A_TARGET_POSITION;
	   OP10A_SRV_RH_BDYGRP_STUS.moveAbsolute	:= OP10A_MOVE_TARGET;
	   OP10A_SRV_ACT_POS						:= OP10A_SRV_RH_BDYGRP_STUS.actualPosition;
	   OP10A_SRV_FAULT							:= OP10A_RH_GRIPR.bAxisError;
	   OP10A_SRV_ENABLE							:= OP10A_RH_GRIPR.bAxisEnabled;
	                                			
	5: OP10A_SRV_LH_BDYANG_STUS.jogPos			:= OP10_JOG_POSITIVE AND NOT OP10_JOG_NEGATIVE;
	   OP10A_SRV_LH_BDYANG_STUS.jogNeg   		:= OP10_JOG_NEGATIVE AND NOT OP10_JOG_POSITIVE;
	   OP10A_SRV_LH_BDYANG_CNT.Axis_Home_Cmd	:= OP10A_SET_HOME;
	   OP10A_SRV_LH_BDYANG_STUS.targetPositon	:= OP10A_TARGET_POSITION;
	   OP10A_SRV_LH_BDYANG_STUS.moveAbsolute	:= OP10A_MOVE_TARGET;
	   OP10A_SRV_ACT_POS						:= OP10A_SRV_LH_BDYANG_STUS.actualPosition;
	   OP10A_SRV_FAULT							:= OP10A_LH_ROTY.bAxisError;
	   OP10A_SRV_ENABLE							:= OP10A_LH_ROTY.bAxisEnabled;
                                			
	6: OP10A_SRV_RH_BDYANG_STUS.jogPos			:= OP10_JOG_POSITIVE AND NOT OP10_JOG_NEGATIVE;
	   OP10A_SRV_RH_BDYANG_STUS.jogNeg   		:= OP10_JOG_NEGATIVE AND NOT OP10_JOG_POSITIVE;
	   OP10A_SRV_RH_BDYANG_CNT.Axis_Home_Cmd	:= OP10A_SET_HOME;
	   OP10A_SRV_RH_BDYANG_STUS.targetPositon	:= OP10A_TARGET_POSITION;
	   OP10A_SRV_RH_BDYANG_STUS.moveAbsolute	:= OP10A_MOVE_TARGET;
	   OP10A_SRV_ACT_POS						:= OP10A_SRV_RH_BDYANG_STUS.actualPosition;
	   OP10A_SRV_FAULT							:= OP10A_RH_ROTY.bAxisError;
	   OP10A_SRV_ENABLE							:= OP10A_RH_ROTY.bAxisEnabled;
                           			
	11:OP10_SRV_FRST_PCKBDY_STUS.jogPos			:= OP10_JOG_POSITIVE AND NOT OP10_JOG_NEGATIVE;
	   OP10_SRV_FRST_PCKBDY_STUS.jogNeg  		:= OP10_JOG_NEGATIVE AND NOT OP10_JOG_POSITIVE;
	   OP10_SRV_FRST_PCKBDY_CNT.Axis_Home_Cmd	:= OP10A_SET_HOME;
	   OP10_SRV_FRST_PCKBDY_STUS.targetPositon	:= OP10A_TARGET_POSITION;    
	   OP10_SRV_FRST_PCKBDY_STUS.moveAbsolute	:= OP10A_MOVE_TARGET;
	   OP10A_SRV_ACT_POS						:= OP10_SRV_FRST_PCKBDY_STUS.actualPosition;
	   OP10A_SRV_FAULT							:= OP10_FRT_BDY_GPR.bAxisError;
	   OP10A_SRV_ENABLE							:= OP10_FRT_BDY_GPR.bAxisEnabled;

                         			
	12:OP10_SRV_SCND_PCKBDY_STUS.jogPos			:= OP10_JOG_POSITIVE AND NOT OP10_JOG_NEGATIVE;
	   OP10_SRV_SCND_PCKBDY_STUS.jogNeg  		:= OP10_JOG_NEGATIVE AND NOT OP10_JOG_POSITIVE;   
	   OP10_SRV_SCND_PCKBDY_CNT.Axis_Home_Cmd	:= OP10A_SET_HOME;
	   OP10_SRV_SCND_PCKBDY_STUS.targetPositon	:= OP10A_TARGET_POSITION;
	   OP10_SRV_SCND_PCKBDY_STUS.moveAbsolute	:= OP10A_MOVE_TARGET;
	   OP10A_SRV_ACT_POS						:= OP10_SRV_SCND_PCKBDY_STUS.actualPosition;
	   OP10A_SRV_FAULT							:= OP10_SEC_BDY_GPR.bAxisError;
	   OP10A_SRV_ENABLE							:= OP10_SEC_BDY_GPR.bAxisEnabled;	   
END_CASE

ELSE
		OP10_CYL_NO									:=0;	
		OP10A_O_HORZ_MANUALPB1						:=FALSE;
		OP10A_O_HORZ_MANUALPB2						:=FALSE;
		OP10A_O_VERT_MANUALPB1						:=FALSE;
		OP10A_O_VERT_MANUALPB2						:=FALSE;
		OP10A_M_O_LHGRIP_ONOFF						:=FALSE;
		OP10A_O_0DEGRE_MANUALPB1					:=FALSE;
		OP10A_O_180DEGRE_MANUALPB2					:=FALSE;
		OP10A_M_O_LHPUSH_CYL						:=FALSE;
		OP10A_M_LNR1_ONOFF		    				:=FALSE;
		OP10A_M_LNR2_ONOFF          				:=FALSE;
		OP10A_M_BOWL_ONOFF         					:=FALSE;
		OP10A_M_HOPPER_ONOFF       					:=FALSE;
		OP10A_M_O_RHPUSH_CYL						:=FALSE;	
		OP10A_M_O_RHGRIP_ONOFF						:=FALSE;
		OP10A_M_RH_REJ_HOME							:=FALSE;
		OP10A_M_RH_REJ_WRK	 						:=FALSE;
		OP10A_M_LH_REJ_HOME							:=FALSE;
		OP10A_M_LH_REJ_WRK	 						:=FALSE;		
		OP10_FRT_BDY_SING_HME	 					:=FALSE;
		OP10_FRT_BDY_SING_WRK						:=FALSE;
		OP10_SEC_BDY_SING_HME	 					:=FALSE;
		OP10_SEC_BDY_SING_WRK						:=FALSE;		
		
		
		
END_IF
	

//#############################		OP10B		###############################



IF OP10B_MANUAL_SELECTED THEN
//OP10B                         				
	OP10B_M_LNR1_ONOFF          				:= OP10B_H_LNR1_ONOFF  ;
	OP10B_M_LNR2_ONOFF          				:= OP10B_H_LNR2_ONOFF  ;
	OP10B_M_BOWL_ONOFF          				:= OP10B_H_BOWL_ONOFF  ;
	OP10B_M_HOPPER_ONOFF        				:= OP10B_H_HOPPER_ONOFF;	

CASE OP10B_CYL_NO OF 

5: IF OP10B_HOME THEN            		
		OP10B_O_HORZ_MANUALPB1					:=TRUE;
		OP10B_O_HORZ_MANUALPB2					:=FALSE;
		END_IF                      			
		IF OP10B_WORK THEN           			
		OP10B_O_HORZ_MANUALPB1					:=FALSE;
		OP10B_O_HORZ_MANUALPB2					:=TRUE;
		END_IF                      			
                                    			
	6: IF OP10B_HOME THEN            			
		OP10B_O_VERT_MANUALPB1					:=TRUE;
		OP10B_O_VERT_MANUALPB2					:=FALSE;
		END_IF                      			
		IF OP10B_WORK THEN           			
		OP10B_O_VERT_MANUALPB1					:=FALSE;
		OP10B_O_VERT_MANUALPB2					:=TRUE;
		END_IF                      		
		                            		
	8:IF OP10B_HOME THEN             		
		OP10B_O_0DEGRE_MANUALPB1				:=TRUE;
		OP10B_O_180DEGRE_MANUALPB2				:=FALSE;
		END_IF                      			
		IF OP10B_WORK THEN           			
		OP10B_O_0DEGRE_MANUALPB1				:=FALSE;
		OP10B_O_180DEGRE_MANUALPB2				:=TRUE;
		END_IF                              	
	                                        	
	11: IF OP10B_HOME THEN           			
		OP10B_M_LH_REJ_HOME						:=TRUE;
		OP10B_M_LH_REJ_WRK	 	 				:=FALSE;
		END_IF                      		
		IF OP10B_WORK THEN           		
		OP10B_M_LH_REJ_HOME						:=FALSE;
		OP10B_M_LH_REJ_WRK	 					:=TRUE;
		END_IF                      			
                       			            	
	12: IF OP10B_HOME THEN           			
		OP10B_M_RH_REJ_HOME						:=TRUE;
		OP10B_M_RH_REJ_WRK	  	 				:=FALSE;
		END_IF                      			
		IF OP10B_WORK THEN           			
		OP10B_M_RH_REJ_HOME						:=FALSE;
		OP10B_M_RH_REJ_WRK	 					:=TRUE;
		END_IF 	

	17: IF OP10B_HOME THEN           		
		OP10B_M_O_LHGRIP_ONOFF					:=FALSE;
		END_IF                      			
		IF OP10B_WORK THEN           			
		OP10B_M_O_LHGRIP_ONOFF					:=TRUE;
		END_IF                      			
		                            			
	18:	IF OP10B_HOME THEN           			
		OP10B_M_O_RHGRIP_ONOFF					:=FALSE;
		END_IF                      			
		IF OP10B_WORK THEN           			
		OP10B_M_O_RHGRIP_ONOFF					:=TRUE;
		END_IF                      			
		                            			
	19: IF OP10B_HOME THEN           			
		OP10B_M_O_LHPUSH_CYL					:=FALSE;
		END_IF                      		
		IF OP10B_WORK THEN           		
		OP10B_M_O_LHPUSH_CYL					:=TRUE;
		END_IF                      			
		                            			
	20: IF OP10B_HOME THEN           			
		OP10B_M_O_RHPUSH_CYL					:=FALSE;
		END_IF                      			
		IF OP10B_WORK THEN           			
		OP10B_M_O_RHPUSH_CYL					:=TRUE;
		END_IF 

END_CASE	
	
CASE OP10B_SERVO_NO OF 
	
	2: OP10B_SRV_O_CNVY_STUS.jogPos				:= OP10B_JOG_POSITIVE AND NOT OP10B_JOG_NEGATIVE;
	   OP10B_SRV_O_CNVY_STUS.jogNeg				:= OP10B_JOG_NEGATIVE AND NOT OP10B_JOG_POSITIVE;
	   OP10B_SRV_O_CNVY_CNT.Bsethome	        := OP10B_SET_HOME;
	   OP10B_SRV_O_CNVY_STUS.targetPositon	    := OP10B_TARGET_POSITION;
//	   OP10B_SRV_LH_BDYGRP_STUS.targetVelocity	:= OP10B_TARGET_VEL;
	   OP10B_SRV_O_CNVY_STUS.moveAbsolute	    := OP10B_MOVE_TARGET;
	   OP10B_SRV_ACT_POS						:= OP10B_SRV_O_CNVY_STUS.actualPosition;
	   OP10B_SRV_FAULT							:= OP10B_CONVEYOR.bAxisError;
	   OP10B_SRV_ENABLE							:= OP10B_CONVEYOR.bAxisEnabled;
                                    	
	7: OP10B_SRV_LH_BDYGRP_STUS.jogPos			:= OP10B_JOG_POSITIVE AND NOT OP10B_JOG_NEGATIVE;
	   OP10B_SRV_LH_BDYGRP_STUS.jogNeg			:= OP10B_JOG_NEGATIVE AND NOT OP10B_JOG_POSITIVE;
	   OP10B_SRV_LH_BDYGRP_CNT.Axis_Home_Cmd	:= OP10B_SET_HOME;
	   OP10B_SRV_LH_BDYGRP_STUS.targetPositon	:= OP10B_TARGET_POSITION;
//	   OP10B_SRV_LH_BDYGRP_STUS.targetVelocity	:= OP10B_TARGET_VEL;
	   OP10B_SRV_LH_BDYGRP_STUS.moveAbsolute	:= OP10B_MOVE_TARGET;
	   OP10B_SRV_ACT_POS						:= OP10B_SRV_LH_BDYGRP_STUS.actualPosition;
	   OP10B_SRV_FAULT							:= OP10B_LH_GRIPR.bAxisError;
	   OP10B_SRV_ENABLE							:= OP10B_LH_GRIPR.bAxisEnabled;	   
	   
	                                		
	8: OP10B_SRV_RH_BDYGRP_STUS.jogPos			:= OP10B_JOG_POSITIVE AND NOT OP10B_JOG_NEGATIVE;
	   OP10B_SRV_RH_BDYGRP_STUS.jogNeg    		:= OP10B_JOG_NEGATIVE AND NOT OP10B_JOG_POSITIVE;
	   OP10B_SRV_RH_BDYGRP_CNT.Axis_Home_Cmd	:= OP10B_SET_HOME;
	   OP10B_SRV_RH_BDYGRP_STUS.targetPositon	:= OP10B_TARGET_POSITION;
//	   OP10B_SRV_RH_BDYGRP_STUS.targetVelocity	:= OP10B_TARGET_VEL;
	   OP10B_SRV_RH_BDYGRP_STUS.moveAbsolute	:= OP10B_MOVE_TARGET;
	   OP10B_SRV_ACT_POS						:= OP10B_SRV_RH_BDYGRP_STUS.actualPosition;
	   OP10B_SRV_FAULT							:= OP10B_RH_GRIPR.bAxisError;
	   OP10B_SRV_ENABLE							:= OP10B_RH_GRIPR.bAxisEnabled;	
	   
	                                			
	9: OP10B_SRV_LH_BDYANG_STUS.jogPos			:= OP10B_JOG_POSITIVE AND NOT OP10B_JOG_NEGATIVE;
	   OP10B_SRV_LH_BDYANG_STUS.jogNeg   		:= OP10B_JOG_NEGATIVE AND NOT OP10B_JOG_POSITIVE;
	   OP10B_SRV_LH_BDYANG_CNT.Axis_Home_Cmd	:= OP10B_SET_HOME;
	   OP10B_SRV_LH_BDYANG_STUS.targetPositon	:= OP10B_TARGET_POSITION;
//	   OP10B_SRV_LH_BDYANG_STUS.targetVelocity	:= OP10B_TARGET_VEL;
	   OP10B_SRV_LH_BDYANG_STUS.moveAbsolute	:= OP10B_MOVE_TARGET;
	   OP10B_SRV_ACT_POS						:= OP10B_SRV_LH_BDYANG_STUS.actualPosition;
	   OP10B_SRV_FAULT							:= OP10B_LH_ROTY.bAxisError;
	   OP10B_SRV_ENABLE							:= OP10B_LH_ROTY.bAxisEnabled;	   
	                                			
	10:OP10B_SRV_RH_BDYANG_STUS.jogPos			:= OP10B_JOG_POSITIVE AND NOT OP10B_JOG_NEGATIVE;
	   OP10B_SRV_RH_BDYANG_STUS.jogNeg    		:= OP10B_JOG_NEGATIVE AND NOT OP10B_JOG_POSITIVE;
	   OP10B_SRV_RH_BDYANG_CNT.Axis_Home_Cmd	:= OP10B_SET_HOME;
	   OP10B_SRV_RH_BDYANG_STUS.targetPositon	:= OP10B_TARGET_POSITION;
//	   OP10B_SRV_RH_BDYANG_STUS.targetVelocity	:= OP10B_TARGET_VEL;
	   OP10B_SRV_RH_BDYANG_STUS.moveAbsolute	:= OP10B_MOVE_TARGET;
	   OP10B_SRV_ACT_POS						:= OP10B_SRV_RH_BDYANG_STUS.actualPosition;
	   OP10B_SRV_FAULT							:= OP10B_RH_ROTY.bAxisError;
	   OP10B_SRV_ENABLE							:= OP10B_RH_ROTY.bAxisEnabled;	

END_CASE	

ELSE
	OP10B_O_HORZ_MANUALPB1						:=FALSE;		
	OP10B_O_HORZ_MANUALPB2						:=FALSE;		
	OP10B_O_VERT_MANUALPB1						:=FALSE;		
	OP10B_O_VERT_MANUALPB2						:=FALSE;		
	OP10B_M_O_LHGRIP_ONOFF						:=FALSE;		
	OP10B_O_0DEGRE_MANUALPB1					:=FALSE;	
	OP10B_O_180DEGRE_MANUALPB2					:=FALSE;
	OP10B_M_O_LHPUSH_CYL  						:=FALSE;		
	OP10B_M_LNR1_ONOFF  						:=FALSE;		
	OP10B_M_LNR2_ONOFF  						:=FALSE;		
	OP10B_M_BOWL_ONOFF  						:=FALSE;		
	OP10B_M_O_RHPUSH_CYL						:=FALSE;
	OP10B_M_O_RHGRIP_ONOFF						:=FALSE;	
	OP10B_M_RH_REJ_HOME							:=FALSE;
	OP10B_M_RH_REJ_WRK	  	 					:=FALSE;	
	OP10B_M_LH_REJ_HOME							:=FALSE;
	OP10B_M_LH_REJ_WRK	 						:=FALSE;

END_IF
// OP10B_HORZ_CYLINDER_SAFE_WRK/HME
OP10A_HORZ_CYL.SafeHome				:=OP10A_VERT_CYL.Sensor1 ;//AND OP10A_DEGREE_CYL.Sensor1;
OP10A_HORZ_CYL.SafeWork             :=OP10A_VERT_CYL.Sensor1 ;//AND OP10A_DEGREE_CYL.Sensor1;


OP10A_HORZ_CYL(
	Auto:= OP10A_AUTO_RUNNING OR OP10A_STEP_RUNNING OR OP10A_CYL_PNP_CHECK, 
	Manual:= OP10A_MANUAL_SELECTED,
	HOMING_RUNNING:= OP10A_START_HOMNG, 
	ErrorActive:= OP10A_ERR, 
	ResetPB:= Servo_Reset, 								
	Sensor1:= I10A_ORING_HORZ_CYL_REV_I1011_2,         						(*OP10A_HORZ_CYL_FUNTIONAL_BLCK*)                                
	Sensor2:= I10A_ORING_HORZ_CYL_FWD_I1011_3, 
	ManualPB1:= OP10A_O_HORZ_MANUALPB1, 
	ManualPB2:= OP10A_O_HORZ_MANUALPB2, 
	AutoCmd1:= OP10A_O_HORZ_AUTOCMD1, 
	AutoCmd2:= OP10A_O_HORZ_AUTOCMD2, 
	OperationEnable:= OperationEnable, 
	SafeHome:= , 
	SafeWork:= , 
	Pulse_1Sec:= Pulse_Block.Q1Hz, 
	BlinkingBit:= , 
	TimeOut1:= 5, 
	TimeOut2:= 5, 
	TimeOut3:= 5,
	HOMING_STRT:= (OP10A_HME_STP_NO=15), 
	HME_DLY:= 100, 
	HME_DN_NO:= OP10A_HME_15_20, 
	HME_CYL_2:= TRUE, 
	HME_CYL_3:= TRUE, 
	Solenoid1=> O10A_ORING_HORZ_CYL_REV_Q1050_6, 
	Solenoid2=> O10A_ORING_HORZ_CYL_FWD_Q1050_7, 
	AlarmSensor1=> OP10A_HORZ_CYL_A1, 
	AlarmSensor2=> OP10A_HORZ_CYL_A2, 
	AlarmSolenoid1=> OP10A_HORZ_CYL_A3, 
	AlarmSolenoid2=> OP10A_HORZ_CYL_A4, 
	AllSignal=> OP10A_HORZ_CYL_A5, 
	AlarmPresent=> OP10A_CYLINDER_ERR.0, 
	Position1=> , 
	Position2=> , 
	HomeSensorBlink=> , 
	WorkSensorBlink=> ,
	Status:= OP10A_HORZ_CYL_STUS,
	HMENG_RESULT := OP10A_HME_STP_NO);
	

// OP10A_VERT_CYLINDER_SAFE_WRK/HME
OP10A_VERT_CYL.SafeHome				:= OP10A_HORZ_CYL.Sensor1 OR OP10A_HORZ_CYL.Sensor2;
OP10A_VERT_CYL.SafeWork				:= (OP10A_HORZ_CYL.Sensor1 OR OP10A_HORZ_CYL.Sensor2) AND OP10A_DEGREE_CYL.Sensor1;
	
OP10A_VERT_CYL(
	Auto:= OP10A_AUTO_RUNNING OR OP10A_STEP_RUNNING OR OP10A_CYL_PNP_CHECK, 
	Manual:= OP10A_MANUAL_SELECTED,
	HOMING_RUNNING:= OP10A_START_HOMNG, 
	ErrorActive:= OP10A_ERR, 
	ResetPB:= Servo_Reset, 
	Sensor1:= I10A_ORING_VERT_CYL_UP_I1011_4, 
	Sensor2:= I10A_ORING_VERT_CYL_DWN_I1011_5, 								(*OP10A_VERT_CYL_FUNTIONAL_BLOCK*)
	ManualPB1:= OP10A_O_VERT_MANUALPB1, 
	ManualPB2:= OP10A_O_VERT_MANUALPB2, 
	AutoCmd1:= OP10A_O_VERT_AUTOCMD1, 
	AutoCmd2:= OP10A_O_VERT_AUTOCMD2, 
	OperationEnable:= OperationEnable, 
	SafeHome:= , 
	SafeWork:= , 
	Pulse_1Sec:= Pulse_Block.Q1Hz, 
	BlinkingBit:= , 
	TimeOut1:= 5, 
	TimeOut2:= 5, 
	TimeOut3:= 5,
	HOMING_STRT:= (OP10A_HME_STP_NO=20), 
	HME_DLY:= 100, 
	HME_DN_NO:= OP10A_HME_20_25, 
	HME_CYL_2:=TRUE , 
	HME_CYL_3:=TRUE , 
	Solenoid1=> O10A_ORING_VERT_CYL_UP_Q1051_0, 
	Solenoid2=> O10A_ORING_VERT_CYL_DWN_Q1051_1, 
	AlarmSensor1=> OP10A_VERT_CYL_A1, 
	AlarmSensor2=> OP10A_VERT_CYL_A2, 
	AlarmSolenoid1=> OP10A_VERT_CYL_A3, 
	AlarmSolenoid2=> OP10A_VERT_CYL_A4, 
	AllSignal=> OP10A_VERT_CYL_A5, 
	AlarmPresent=> OP10A_CYLINDER_ERR.1, 
	Position1=> , 
	Position2=> , 
	HomeSensorBlink=> , 
	WorkSensorBlink=> ,
	Status:= OP10A_VERT_CYL_STUS,
	HMENG_RESULT := OP10A_HME_STP_NO);

// OP10A_DEGREE_CYLINDER_SAFE_WRK/HME	
OP10A_DEGREE_CYL.SafeHome				:= OP10A_HORZ_CYL.Sensor1 AND OP10A_VERT_CYL.Sensor1;
OP10A_DEGREE_CYL.SafeWork				:= OP10A_HORZ_CYL.Sensor1 AND OP10A_VERT_CYL.Sensor1; 
	
	
OP10A_DEGREE_CYL(
	Auto:= OP10A_AUTO_RUNNING OR OP10A_STEP_RUNNING OR OP10A_CYL_PNP_CHECK, 
	Manual:= OP10A_MANUAL_SELECTED,
	HOMING_RUNNING:= OP10A_START_HOMNG, 
	ErrorActive:= OP10A_ERR, 
	ResetPB:= Servo_Reset, 
	Sensor1:= I10A_ORING_ROTRY_CYL_O_DEG_I1011_0, 							(*OP10A_DEGREE_CYL_FUNTIONAL_BLCK*)
	Sensor2:= I10A_ORING_ROTRY_CYL_180_DEG_I1011_1, 
	ManualPB1:= OP10A_O_0DEGRE_MANUALPB1, 
	ManualPB2:= OP10A_O_180DEGRE_MANUALPB2, 
	AutoCmd1:= OP10A_O_0DEGRE_AUTOCMD1, 
	AutoCmd2:= OP10A_O_180DEGRE_AUTOCMD2, 
	OperationEnable:= OperationEnable, 
	SafeHome:= , 
	SafeWork:= , 
	Pulse_1Sec:= Pulse_Block.Q1Hz, 
	BlinkingBit:= , 
	TimeOut1:= 5, 
	TimeOut2:= 5, 
	TimeOut3:= 5,
	HOMING_STRT:= (OP10A_HME_STP_NO=25), 
	HME_DLY:= 100, 
	HME_DN_NO:=  OP10A_HME_25_30, 
	HME_CYL_2:=TRUE , 
	HME_CYL_3:=TRUE , 
	Solenoid1=> O10A_ORING_ROTRY_CYL_O_DEG_Q1050_4, 
	Solenoid2=> O10A_ORING_ROTRY_CYL_180_DEG_Q1050_5, 
	AlarmSensor1=> OP10A_DEGREE_CYL_A1, 
	AlarmSensor2=> OP10A_DEGREE_CYL_A2, 
	AlarmSolenoid1=> OP10A_DEGREE_CYL_A3, 
	AlarmSolenoid2=> OP10A_DEGREE_CYL_A4, 
	AllSignal=> OP10A_DEGREE_CYL_A5, 
	AlarmPresent=> OP10A_CYLINDER_ERR.2, 
	Position1=> , 
	Position2=> , 
	HomeSensorBlink=> , 
	WorkSensorBlink=> ,
	Status:= OP10A_DEGREE_CYL_STUS,
	HMENG_RESULT := OP10A_HME_STP_NO);
	
// OP10A_LH_GRIPPER_CYLINDER_SAFE_WRK/HME	
OP10A_LH_GRP.SafeHome						:= OP10A_LH_PUSH.Sensor1;
OP10A_LH_GRP.SafeWork						:= OP10A_LH_PUSH.Sensor1;

	
OP10A_LH_GRP(
	Auto:= OP10A_AUTO_RUNNING OR OP10A_STEP_RUNNING OR OP10A_CYL_PNP_CHECK, 
	Manual:= OP10A_MANUAL_SELECTED,
	HOMING_RUNNING:= OP10A_START_HOMNG, 
	ErrorActive:= OP10A_ERR, 
	ResetPB:= Servo_Reset, 
	Sensor1:= I10A_ORING_LH_GRPR_CLSE_I1010_2, 								(*OP10A_LH_GRIPPER_FUNCATIONAL_BLOCK*)
	Sensor2:= I10A_ORING_LH_GRPR_OPN_I1010_3, 
	ManualPB1:=OP10A_LH_GRP.Manual AND  NOT OP10A_M_O_LHGRIP_ONOFF,//NOT OP10A_M_O_LHGRIP_ONOFF, 
	ManualPB2:=OP10A_LH_GRP.Manual AND OP10A_M_O_LHGRIP_ONOFF,//OP10A_M_O_LHGRIP_ONOFF, 
	AutoCmd1:=OP10A_LH_GRP.Auto AND NOT OP10A_A_O_LHGRIP_ONOFF,// NOT OP10A_A_O_LHGRIP_ONOFF, 
	AutoCmd2:=OP10A_LH_GRP.Auto AND OP10A_A_O_LHGRIP_ONOFF, 
	OperationEnable:= OperationEnable, 
	SafeHome:= 1, 
	SafeWork:= 1, 
	Pulse_1Sec:= Pulse_Block.Q1Hz, 
	BlinkingBit:= , 
	TimeOut1:= 5, 
	TimeOut2:= 5, 
	TimeOut3:= 5,
	HOMING_STRT:=(OP10A_HME_STP_NO=5), 
	HME_DLY:= 100, 
	HME_DN_NO:= OP10A_HME_5_10, 
	HME_CYL_2:= OP10A_RH_GRP.Sensor1, 
	HME_CYL_3:=TRUE , 
	Solenoid1=> , 
	Solenoid2=>O10A_ORING_LH_GRPR_CLSE_OPN_Q1050_0 , 
	AlarmSensor1=> OP10A_LH_GRP_A1, 
	AlarmSensor2=> OP10A_LH_GRP_A2, 
	AlarmSolenoid1=> OP10A_LH_GRP_A3, 
	AlarmSolenoid2=> OP10A_LH_GRP_A4, 
	AllSignal=> OP10A_LH_GRP_A5, 
	AlarmPresent=> OP10A_CYLINDER_ERR.3, 
	Position1=> , 
	Position2=> , 
	HomeSensorBlink=> , 
	WorkSensorBlink=> ,	
	Status:= OP10A_LH_GRP_STATS,
	HMENG_RESULT := OP10A_HME_STP_NO);

// OP10A_RH_GRIPPER_CYLINDER_SAFE_WRK/HME	
OP10A_RH_GRP.SafeHome						:= OP10A_RH_PUSH.Sensor1;
OP10A_RH_GRP.SafeWork						:= OP10A_RH_PUSH.Sensor1;				// CHANGE THE INPUT AS FALSE

	
	
OP10A_RH_GRP(
	Auto:= OP10A_AUTO_RUNNING OR OP10A_STEP_RUNNING OR OP10A_CYL_PNP_CHECK, 
	Manual:= OP10A_MANUAL_SELECTED,
	HOMING_RUNNING:= OP10A_START_HOMNG, 
	ErrorActive:= OP10A_ERR, 
	ResetPB:= Servo_Reset, 
	Sensor1:= I10A_ORING_RH_GRPR_CLSE_I1010_6, 
	Sensor2:= I10A_ORING_RH_GRPR_OPN_I1010_5, 
	ManualPB1:=OP10A_RH_GRP.Manual AND  NOT OP10A_M_O_RHGRIP_ONOFF, 
	ManualPB2:= OP10A_RH_GRP.Manual AND OP10A_M_O_RHGRIP_ONOFF, 									(*OP10A_RH_GRIPPER_CYLINDER*)
	AutoCmd1:=OP10A_RH_GRP.Auto AND NOT OP10A_A_O_RHGRIP_ONOFF, 
	AutoCmd2:=OP10A_RH_GRP.Auto AND OP10A_A_O_RHGRIP_ONOFF, 
	OperationEnable:= OperationEnable, 
	SafeHome:= 1, 
	SafeWork:= 1, 
	Pulse_1Sec:= Pulse_Block.Q1Hz, 
	BlinkingBit:= , 
	TimeOut1:= 5, 
	TimeOut2:= 5, 
	TimeOut3:= 5,
	HOMING_STRT:= (OP10A_HME_STP_NO=5),
	HME_DLY:= ,
	HME_DN_NO:= ,
	HME_CYL_2:=TRUE ,
	HME_CYL_3:=TRUE , 
	Solenoid1=> , 
	Solenoid2=> O10A_ORING_RH_GRPR_CLSE_OPN_Q1050_2, 
	AlarmSensor1=> OP10A_RH_GRP_A1, 
	AlarmSensor2=> OP10A_RH_GRP_A2, 
	AlarmSolenoid1=> OP10A_RH_GRP_A3, 
	AlarmSolenoid2=> OP10A_RH_GRP_A4, 
	AllSignal=> OP10A_RH_GRP_A5, 
	AlarmPresent=> OP10A_CYLINDER_ERR.4, 
	Position1=> , 
	Position2=> , 
	HomeSensorBlink=> , 
	WorkSensorBlink=> ,	
	Status:= OP10A_RH_GRP_STUS,
	HMENG_RESULT := OP10A_PARALLEL);

// OP10A_LH_PUSH_CYLINDER_SAFE_WRK/HME
OP10A_LH_PUSH.SafeHome						:=OP10A_LH_GRP.Sensor2 ;
OP10A_LH_PUSH.SafeWork						:=OP10A_LH_GRP.Sensor2 ;

	
OP10A_LH_PUSH(
	Auto:= OP10A_AUTO_RUNNING OR OP10A_STEP_RUNNING OR OP10A_CYL_PNP_CHECK, 
	Manual:= OP10A_MANUAL_SELECTED,
	HOMING_RUNNING:= OP10A_START_HOMNG, 
	ErrorActive:= OP10A_ERR, 
	ResetPB:= Servo_Reset, 
	Sensor1:= NOT I10A_ORING_LH_PUSHR_CYL_REV_I1010_4, 										(*OP10A_LH_PUSHING_CYLINDER*)
	Sensor2:= I10A_ORING_LH_PUSHR_CYL_REV_I1010_4, 
	ManualPB1:=OP10A_LH_PUSH.Manual AND NOT OP10A_M_O_LHPUSH_CYL, 
	ManualPB2:=OP10A_LH_PUSH.Manual AND OP10A_M_O_LHPUSH_CYL, 
	AutoCmd1:=OP10A_LH_PUSH.Auto AND NOT OP10A_A_O_LHPUSH_CYL, 
	AutoCmd2:=OP10A_LH_PUSH.Auto AND OP10A_A_O_LHPUSH_CYL, 
	OperationEnable:= OperationEnable, 
	SafeHome:= , 
	SafeWork:= , 
	Pulse_1Sec:= Pulse_Block.Q1Hz, 
	BlinkingBit:= , 
	TimeOut1:= 5, 
	TimeOut2:= 5, 
	TimeOut3:= 5,
	HOMING_STRT:= (OP10A_HME_STP_NO=1),
	HME_DLY:= 100,
	HME_DN_NO:= OP10A_HME_1_5,
	HME_CYL_2:= OP10A_RH_PUSH.Sensor1,
	HME_CYL_3:=TRUE , 
	Solenoid1=> , 
	Solenoid2=> O10A_ORING_LH_PUSHR_CYL_REV_FWD_Q1050_1, 
	AlarmSensor1=> OP10A_LH_PUSH_A1, 
	AlarmSensor2=> OP10A_LH_PUSH_A2, 
	AlarmSolenoid1=> OP10A_LH_PUSH_A3, 
	AlarmSolenoid2=> OP10A_LH_PUSH_A4, 
	AllSignal=> OP10A_LH_PUSH_A5, 
	AlarmPresent=> OP10A_CYLINDER_ERR.5, 
	Position1=> , 
	Position2=> , 
	HomeSensorBlink=> , 
	WorkSensorBlink=> ,	
	Status:= OP10A_LH_PUSH_STUS,
	HMENG_RESULT := OP10A_HME_STP_NO);


// OP10A_LH_PUSH_CYLINDER_SAFE_WRK/HME
OP10A_RH_PUSH.SafeHome						:= OP10A_RH_GRP.Sensor2 ;
OP10A_RH_PUSH.SafeWork						:= OP10A_RH_GRP.Sensor2 ;


OP10A_RH_PUSH(
	Auto:= OP10A_AUTO_RUNNING OR OP10A_STEP_RUNNING OR OP10A_CYL_PNP_CHECK, 
	Manual:= OP10A_MANUAL_SELECTED,
	HOMING_RUNNING:= OP10A_START_HOMNG, 
	ErrorActive:= OP10A_ERR, 								(*OP10A_RH _ PUSHING CYL_FUNTIONAL_BLCK*)
	ResetPB:= Servo_Reset, 
	Sensor1:= NOT I10A_ORING_RH_PUSHR_CYL_REV_I1010_7, 
	Sensor2:=I10A_ORING_RH_PUSHR_CYL_REV_I1010_7 , 
	ManualPB1:=OP10A_RH_PUSH.Manual AND NOT OP10A_M_O_RHPUSH_CYL, 
	ManualPB2:=OP10A_RH_PUSH.Manual AND OP10A_M_O_RHPUSH_CYL, 
	AutoCmd1:=OP10A_RH_PUSH.AUTO AND NOT OP10A_A_O_RHPUSH_CYL, 
	AutoCmd2:= OP10A_RH_PUSH.AUTO AND OP10A_A_O_RHPUSH_CYL, 
	OperationEnable:= OperationEnable, 
	SafeHome:= , 
	SafeWork:= , 
	Pulse_1Sec:= Pulse_Block.Q1Hz, 
	BlinkingBit:= , 
	TimeOut1:= 5, 
	TimeOut2:= 5, 
	TimeOut3:= 5,
	HOMING_STRT:= (OP10A_HME_STP_NO=1),
	HME_DLY:= ,
	HME_DN_NO:= ,
	HME_CYL_2:=TRUE ,
	HME_CYL_3:=TRUE , 
	Solenoid1=> , 
	Solenoid2=>O10A_ORING_RH_PUSHR_CYL_REV_FWD_Q1050_3 , 
	AlarmSensor1=> OP10A_RH_PUSH_A1, 
	AlarmSensor2=> OP10A_RH_PUSH_A2, 
	AlarmSolenoid1=> OP10A_RH_PUSH_A3, 
	AlarmSolenoid2=> OP10A_RH_PUSH_A4, 
	AllSignal=> OP10A_RH_PUSH_A5, 
	AlarmPresent=> OP10A_CYLINDER_ERR.6, 
	Position1=> , 
	Position2=> , 
	HomeSensorBlink=> , 
	WorkSensorBlink=> ,	
	Status:= OP10A_RH_PUSH_STUS,
	HMENG_RESULT := OP10A_PARALLEL);
	
// OP10A_LH_REJ_CYLINDER_SAFE_WRK/HME
//OP10A_LH_REJ.SafeHome						:= TRUE;
//OP10A_LH_REJ.SafeWork						:= TRUE;

OP10A_LH_REJ(
	Auto:= OP10A_AUTO_RUNNING OR OP10A_STEP_RUNNING OR OP10A_CYL_PNP_CHECK, 
	Manual:= OP10A_MANUAL_SELECTED,
	HOMING_RUNNING:= OP10A_START_HOMNG, 
	ErrorActive:= OP10A_ERR, 								(*OP10A_RH _ PUSHING CYL_FUNTIONAL_BLCK*)
	ResetPB:= Servo_Reset, 
	Sensor1:= I10A_LH_FIRTRE_ORING_REJ_CYL_REV_I1011_6, 
	Sensor2:= I10A_LH_FIRTRE_ORING_REJ_CYL_FWD_I1011_7 , 
	ManualPB1:= OP10A_M_LH_REJ_HOME, 
	ManualPB2:= OP10A_M_LH_REJ_WRK, 
	AutoCmd1:= OP10A_A_LH_REJ_HOME, 
	AutoCmd2:= OP10A_A_LH_REJ_WRK, 
	OperationEnable:= OperationEnable, 
	SafeHome:= 1, 
	SafeWork:= 1, 
	Pulse_1Sec:= Pulse_Block.Q1Hz, 
	BlinkingBit:= , 
	TimeOut1:= 5, 
	TimeOut2:= 5, 
	TimeOut3:= 5,
	HOMING_STRT:= (OP10A_HME_STP_NO=1),
	HME_DLY:= ,
	HME_DN_NO:= ,
	HME_CYL_2:=TRUE ,
	HME_CYL_3:=TRUE , 
	Solenoid1=>O10A_LH_FIRTRE_ORING_REJ_CYL_REV_Q1051_2 , 
	Solenoid2=>O10A_LH_FIRTRE_ORING_REJ_CYL_FWD_Q1051_3 , 						
	AlarmSensor1=> OP10A_LH_REJ_A1,                    
	AlarmSensor2=> OP10A_LH_REJ_A2,                    
	AlarmSolenoid1=>OP10A_LH_REJ_A3,                   
	AlarmSolenoid2=> OP10A_LH_REJ_A4, 
	AllSignal=> OP10A_LH_REJ_A5, 
	AlarmPresent=> OP10A_CYLINDER_ERR.7, 
	Position1=> , 
	Position2=> , 
	HomeSensorBlink=> , 
	WorkSensorBlink=> ,	
	Status:= OP10A_RH_PUSH_STUS,
	HMENG_RESULT := OP10A_PARALLEL);	
	
// OP10A_RH_REJ_CYLINDER_SAFE_WRK/HME
//OP10A_RH_REJ.SafeHome						:= TRUE;
//OP10A_RH_REJ.SafeWork						:= TRUE;

OP10A_RH_REJ(
	Auto:= OP10A_AUTO_RUNNING OR OP10A_STEP_RUNNING OR OP10A_CYL_PNP_CHECK, 
	Manual:= OP10A_MANUAL_SELECTED,
	HOMING_RUNNING:= OP10A_START_HOMNG, 
	ErrorActive:= OP10A_ERR, 								(*OP10A_RH _ PUSHING CYL_FUNTIONAL_BLCK*)
	ResetPB:= Servo_Reset, 
	Sensor1:= I10A_RH_FIRTRE_ORING_REJ_CYL_REV_I1020_0, 
	Sensor2:= I10A_RH_FIRTRE_ORING_REJ_CYL_FWD_I1020_1, 
	ManualPB1:= OP10A_M_RH_REJ_HOME, 
	ManualPB2:= OP10A_M_RH_REJ_WRK, 
	AutoCmd1:= OP10A_A_RH_REJ_HOME, 
	AutoCmd2:= OP10A_A_RH_REJ_WRK, 
	OperationEnable:= OperationEnable, 
	SafeHome:= 1, 
	SafeWork:= 1, 
	Pulse_1Sec:= Pulse_Block.Q1Hz, 
	BlinkingBit:= , 
	TimeOut1:= 5, 
	TimeOut2:= 5, 
	TimeOut3:= 5,
	HOMING_STRT:= (OP10A_HME_STP_NO=1),
	HME_DLY:= ,
	HME_DN_NO:= ,
	HME_CYL_2:=TRUE ,
	HME_CYL_3:=TRUE , 
	Solenoid1=>O10A_RH_FIRTRE_ORING_REJ_CYL_REV_Q1051_4 , 
	Solenoid2=>O10A_RH_FIRTRE_ORING_REJ_CYL_FWD_Q1051_5 , 
	AlarmSensor1=>  OP10A_RH_REJ_A1,	
	AlarmSensor2=>  OP10A_RH_REJ_A2,	
	AlarmSolenoid1=>OP10A_RH_REJ_A3,	 
	AlarmSolenoid2=> OP10A_RH_REJ_A4, 
	AllSignal=>  OP10A_RH_REJ_A5,	
	AlarmPresent=> OP10A_CYLINDER_ERR.8, 
	Position1=> , 
	Position2=> , 
	HomeSensorBlink=> , 
	WorkSensorBlink=> ,	
	Status:= OP10A_RH_PUSH_STUS,
	HMENG_RESULT := OP10A_PARALLEL);	




////////////////////////////////////OP10B_CYLINDER_BLOCK////////////////////////////////////
// OP10B_HORZ_CYLINDER_SAFE_WRK/HME
OP10B_HORZ_CYL.SafeHome				:=OP10B_VERT_CYL.Sensor1 ;//AND OP10B_DEGREE_CYL.Sensor1;
OP10B_HORZ_CYL.SafeWork             :=OP10B_VERT_CYL.Sensor1 ;//AND OP10B_DEGREE_CYL.Sensor1;

OP10B_HORZ_CYL(
	Auto:= OP10B_AUTO_RUNNING OR OP10B_STEP_RUNNING OR OP10B_CYL_PNP_CHECK , 
	Manual:= OP10B_MANUAL_SELECTED,
	HOMING_RUNNING:= OP10B_START_HOMNG, 
	ErrorActive:= OP10B_ERR, 
	ResetPB:= Servo_Reset, 								
	Sensor1:= I10B_ORING_HORZ_CYL_REV_I1031_2,         						(*OP10B_HORZ_CYL_FUNTIONAL_BLCK*)                                
	Sensor2:= I10B_ORING_HORZ_CYL_FWD_I1031_3, 
	ManualPB1:= OP10B_O_HORZ_MANUALPB1, 
	ManualPB2:= OP10B_O_HORZ_MANUALPB2, 
	AutoCmd1:= OP10B_O_HORZ_AUTOCMD1, 
	AutoCmd2:= OP10B_O_HORZ_AUTOCMD2, 
	OperationEnable:= OperationEnable, 
	SafeHome:=, 
	SafeWork:=, 
	Pulse_1Sec:= Pulse_Block.Q1Hz, 
	BlinkingBit:= , 
	TimeOut1:= 5, 
	TimeOut2:= 5, 
	TimeOut3:= 5,
	HOMING_STRT:= (OP10B_HME_STP_NO= 15),
	HME_DLY:= 100,
	HME_DN_NO:= OP10B_HME_15_20,	
	HME_CYL_2:=TRUE ,
	HME_CYL_3:=TRUE , 
	Solenoid1=> O10B_ORING_HORZ_CYL_REV_Q1060_6, 
	Solenoid2=> O10B_ORING_HORZ_CYL_FWD_Q1060_7, 
	AlarmSensor1=> OP10B_HORZ_CYL_A1, 
	AlarmSensor2=> OP10B_HORZ_CYL_A2, 
	AlarmSolenoid1=> OP10B_HORZ_CYL_A3, 
	AlarmSolenoid2=> OP10B_HORZ_CYL_A4, 
	AllSignal=> OP10B_HORZ_CYL_A5, 
	AlarmPresent=> OP10B_CYLINDER_ERR.0, 
	Position1=> , 
	Position2=> , 
	HomeSensorBlink=> , 
	WorkSensorBlink=> ,	
	Status:= OP10B_HORZ_CYL_STUS,
	HMENG_RESULT := OP10B_HME_STP_NO);
	

// OP10B_VERT_CYLINDER_SAFE_WRK/HME
OP10B_VERT_CYL.SafeHome				:= OP10B_HORZ_CYL.Sensor1 OR OP10B_HORZ_CYL.Sensor2;
OP10B_VERT_CYL.SafeWork				:= (OP10B_HORZ_CYL.Sensor1 OR OP10B_HORZ_CYL.Sensor2) AND OP10B_DEGREE_CYL.Sensor1;
	
OP10B_VERT_CYL(
	Auto:= OP10B_AUTO_RUNNING OR OP10B_STEP_RUNNING OR OP10B_CYL_PNP_CHECK , 
	Manual:= OP10B_MANUAL_SELECTED,
	HOMING_RUNNING:= OP10B_START_HOMNG, 
	ErrorActive:= OP10B_ERR, 
	ResetPB:= Servo_Reset, 
	Sensor1:= I10B_ORING_VERT_CYL_UP_I1031_4, 
	Sensor2:= I10B_ORING_VERT_CYL_DWN_I1031_5, 								(*OP10B_VERT_CYL_FUNTIONAL_BLOCK*)
	ManualPB1:= OP10B_O_VERT_MANUALPB1, 
	ManualPB2:= OP10B_O_VERT_MANUALPB2, 
	AutoCmd1:= OP10B_O_VERT_AUTOCMD1, 
	AutoCmd2:= OP10B_O_VERT_AUTOCMD2, 
	OperationEnable:= OperationEnable, 
	SafeHome:= , 
	SafeWork:= , 
	Pulse_1Sec:= Pulse_Block.Q1Hz, 
	BlinkingBit:= , 
	TimeOut1:= 5, 
	TimeOut2:= 5, 
	TimeOut3:= 5,
	HOMING_STRT:= (OP10B_HME_STP_NO= 20),
	HME_DLY:= 100,
	HME_DN_NO:= OP10B_HME_20_25,
	HME_CYL_2:=TRUE ,
	HME_CYL_3:=TRUE , 
	Solenoid1=> O10B_ORING_VERT_CYL_UP_Q1061_0, 
	Solenoid2=> O10B_ORING_VERT_CYL_DWN_Q1061_1, 
	AlarmSensor1=> OP10B_VERT_CYL_A1, 
	AlarmSensor2=> OP10B_VERT_CYL_A2, 
	AlarmSolenoid1=> OP10B_VERT_CYL_A3, 
	AlarmSolenoid2=> OP10B_VERT_CYL_A4, 
	AllSignal=> OP10B_VERT_CYL_A5, 
	AlarmPresent=> OP10B_CYLINDER_ERR.1, 
	Position1=> , 
	Position2=> , 
	HomeSensorBlink=> , 
	WorkSensorBlink=> ,
	Status:= OP10B_VERT_CYL_STUS,
	HMENG_RESULT := OP10B_HME_STP_NO);

// OP10B_DEGREE_CYLINDER_SAFE_WRK/HME	
OP10B_DEGREE_CYL.SafeHome				:= OP10B_HORZ_CYL.Sensor1 AND OP10B_VERT_CYL.Sensor1;
OP10B_DEGREE_CYL.SafeWork				:= OP10B_HORZ_CYL.Sensor1 AND OP10B_VERT_CYL.Sensor1; 	
	
OP10B_DEGREE_CYL(
	Auto:= OP10B_AUTO_RUNNING OR OP10B_STEP_RUNNING OR OP10B_CYL_PNP_CHECK , 
	Manual:= OP10B_MANUAL_SELECTED,
	HOMING_RUNNING:= OP10B_START_HOMNG, 
	ErrorActive:= OP10B_ERR, 
	ResetPB:= Servo_Reset, 
	Sensor1:= I10B_ORING_ROTRY_CYL_O_DEG_I1031_0, 							(*OP10B_DEGREE_CYL_FUNTIONAL_BLCK*)
	Sensor2:= I10B_ORING_ROTRY_CYL_180_DEG_I1031_1, 
	ManualPB1:= OP10B_O_0DEGRE_MANUALPB1, 
	ManualPB2:= OP10B_O_180DEGRE_MANUALPB2, 
	AutoCmd1:= OP10B_O_0DEGRE_AUTOCMD1, 
	AutoCmd2:= OP10B_O_180DEGRE_AUTOCMD2, 
	OperationEnable:= OperationEnable, 
	SafeHome:=, 
	SafeWork:=, 
	Pulse_1Sec:= Pulse_Block.Q1Hz, 
	BlinkingBit:= , 
	TimeOut1:= 5, 
	TimeOut2:= 5, 
	TimeOut3:= 5,
	HOMING_STRT:= (OP10B_HME_STP_NO= 25),
	HME_DLY:= 100,
	HME_DN_NO:=  OP10B_HME_25_30,
	HME_CYL_2:=TRUE ,
	HME_CYL_3:=TRUE , 
	Solenoid1=> O10B_ORING_ROTRY_CYL_O_DEG_Q1060_4, 
	Solenoid2=> O10B_ORING_ROTRY_CYL_180_DEG_Q1060_5, 
	AlarmSensor1=> OP10B_DEGREE_CYL_A1, 
	AlarmSensor2=> OP10B_DEGREE_CYL_A2, 
	AlarmSolenoid1=> OP10B_DEGREE_CYL_A3, 
	AlarmSolenoid2=> OP10B_DEGREE_CYL_A4, 
	AllSignal=> OP10B_DEGREE_CYL_A5, 
	AlarmPresent=> OP10B_CYLINDER_ERR.2, 
	Position1=> , 
	Position2=> , 
	HomeSensorBlink=> , 
	WorkSensorBlink=> ,	
	Status:= OP10B_DEGREE_CYL_STUS,
	HMENG_RESULT := OP10B_HME_STP_NO);
// OP10B_LH_GRIPPER_CYLINDER_SAFE_WRK/HME	
OP10B_LH_GRP.SafeHome						:= OP10B_LH_PUSH.Sensor1;
OP10B_LH_GRP.SafeWork						:= OP10B_LH_PUSH.Sensor1;

OP10B_LH_GRP(
	Auto:= OP10B_AUTO_RUNNING OR OP10B_STEP_RUNNING OR OP10B_CYL_PNP_CHECK , 
	Manual:= OP10B_MANUAL_SELECTED,
	HOMING_RUNNING:= OP10B_START_HOMNG, 
	ErrorActive:= OP10B_ERR, 
	ResetPB:= Servo_Reset, 
	Sensor1:= I10B_ORING_LH_GRPR_CLSE_I1030_2, 								(*OP10B_LH_GRIPPER_FUNCATIONAL_BLOCK*)
	Sensor2:= I10B_ORING_LH_GRPR_OPN_I1030_3, 
	ManualPB1:=OP10B_MANUAL_SELECTED AND NOT OP10B_M_O_LHGRIP_ONOFF , 
	ManualPB2:=OP10B_MANUAL_SELECTED AND OP10B_M_O_LHGRIP_ONOFF, 
	AutoCmd1:=OP10B_LH_GRP.AUTO AND NOT OP10B_A_O_LHGRIP_ONOFF, 
	AutoCmd2:=OP10B_LH_GRP.AUTO AND OP10B_A_O_LHGRIP_ONOFF, 
	OperationEnable:= OperationEnable, 
	SafeHome:=, 
	SafeWork:=, 
	Pulse_1Sec:= Pulse_Block.Q1Hz, 
	BlinkingBit:= , 
	TimeOut1:= 5, 
	TimeOut2:= 5, 
	TimeOut3:= 5,
	HOMING_STRT:= (OP10B_HME_STP_NO= 5),
	HME_DLY:= 100,
	HME_DN_NO:= OP10B_HME_5_10,
	HME_CYL_2:=OP10B_RH_GRP.Sensor1,
	HME_CYL_3:=TRUE , 
	Solenoid1=> , 
	Solenoid2=> O10B_ORING_LH_GRPR_CLSE_OPN_Q1060_0, 
	AlarmSensor1=> OP10B_LH_GRP_A1, 
	AlarmSensor2=> OP10B_LH_GRP_A2, 
	AlarmSolenoid1=> OP10B_LH_GRP_A3, 
	AlarmSolenoid2=> OP10B_LH_GRP_A4, 
	AllSignal=> OP10B_LH_GRP_A5, 
	AlarmPresent=> OP10B_CYLINDER_ERR.3, 
	Position1=> , 
	Position2=> , 
	HomeSensorBlink=> , 
	WorkSensorBlink=> ,	
	Status:= OP10B_LH_GRP_STATS,
	HMENG_RESULT := OP10B_HME_STP_NO);

// OP10B_RH_GRIPPER_CYLINDER_SAFE_WRK/HME	
OP10B_RH_GRP.SafeHome						:= OP10B_RH_PUSH.Sensor1;
OP10B_RH_GRP.SafeWork						:= OP10B_RH_PUSH.Sensor1;				// CHANGE THE INPUT AS FALSE

OP10B_RH_GRP(
	Auto:= OP10B_AUTO_RUNNING OR OP10B_STEP_RUNNING OR OP10B_CYL_PNP_CHECK  , 
	Manual:= OP10B_MANUAL_SELECTED,
	HOMING_RUNNING:= OP10B_START_HOMNG, 
	ErrorActive:= OP10B_ERR, 
	ResetPB:= Servo_Reset, 
	Sensor1:=I10B_ORING_RH_GRPR_CLSE_I1030_6 , 
	Sensor2:=I10B_ORING_RH_GRPR_OPN_I1030_5 , 
	ManualPB1:=OP10B_MANUAL_SELECTED AND NOT OP10B_M_O_RHGRIP_ONOFF, 
	ManualPB2:=OP10B_MANUAL_SELECTED AND OP10B_M_O_RHGRIP_ONOFF, 									(*OP10B_RH_GRIPPER_CYLINDER*)
	AutoCmd1:=OP10B_RH_GRP.AUTO AND NOT OP10B_A_O_RHGRIP_ONOFF, 
	AutoCmd2:=OP10B_RH_GRP.AUTO AND OP10B_A_O_RHGRIP_ONOFF, 
	OperationEnable:= OperationEnable, 
	SafeHome:= , 
	SafeWork:= , 
	Pulse_1Sec:= Pulse_Block.Q1Hz, 
	BlinkingBit:= , 
	TimeOut1:= 5, 
	TimeOut2:= 5, 
	TimeOut3:= 5,
	HOMING_STRT:= (OP10B_HME_STP_NO= 5),
	HME_DLY:= 100,
	HME_DN_NO:= ,
	HME_CYL_2:=TRUE ,
	HME_CYL_3:=TRUE , 
	Solenoid1=> , 
	Solenoid2=> O10B_ORING_RH_GRPR_CLSE_OPN_Q1060_2, 
	AlarmSensor1=> OP10B_RH_GRP_A1, 
	AlarmSensor2=> OP10B_RH_GRP_A2, 
	AlarmSolenoid1=> OP10B_RH_GRP_A3, 
	AlarmSolenoid2=> OP10B_RH_GRP_A4, 
	AllSignal=> OP10B_RH_GRP_A5, 
	AlarmPresent=> OP10B_CYLINDER_ERR.4, 
	Position1=> , 
	Position2=> , 
	HomeSensorBlink=> , 
	WorkSensorBlink=> ,	
	Status:= OP10B_RH_GRP_STUS,
	HMENG_RESULT := OP10B_PARLLEL);

// OP10B_LH_PUSH_CYLINDER_SAFE_WRK/HME
OP10B_LH_PUSH.SafeHome						:=OP10B_LH_GRP.Sensor2 ;
OP10B_LH_PUSH.SafeWork						:=OP10B_LH_GRP.Sensor2 ;
	
OP10B_LH_PUSH(
	Auto:= OP10B_AUTO_RUNNING OR OP10B_STEP_RUNNING OR OP10B_CYL_PNP_CHECK , 
	Manual:= OP10B_MANUAL_SELECTED,
	HOMING_RUNNING:= OP10B_START_HOMNG, 
	ErrorActive:= OP10B_ERR, 
	ResetPB:= Servo_Reset, 
	Sensor1:= NOT I10B_ORING_LH_PUSHR_CYL_REV_I1030_4, 										(*OP10B_LH_PUSHING_CYLINDER*)
	Sensor2:= I10B_ORING_LH_PUSHR_CYL_REV_I1030_4, 
	ManualPB1:=OP10B_MANUAL_SELECTED AND NOT OP10B_M_O_LHPUSH_CYL, 
	ManualPB2:=OP10B_MANUAL_SELECTED AND OP10B_M_O_LHPUSH_CYL, 
	AutoCmd1:= OP10B_LH_PUSH.AUTO AND NOT OP10B_A_O_LHPUSH_CYL, 
	AutoCmd2:= OP10B_LH_PUSH.AUTO AND OP10B_A_O_LHPUSH_CYL, 
	OperationEnable:= OperationEnable, 
	SafeHome:= 1, 
	SafeWork:= 1, 
	Pulse_1Sec:= Pulse_Block.Q1Hz, 
	BlinkingBit:= , 
	TimeOut1:= 5, 
	TimeOut2:= 5, 
	TimeOut3:= 5,
	HOMING_STRT:= (OP10B_HME_STP_NO= 1),
	HME_DLY:= 100,
	HME_DN_NO:= OP10B_HME_1_5,
	HME_CYL_2:=OP10B_RH_PUSH.Sensor1,
	HME_CYL_3:=TRUE , 
	Solenoid1=> , 
	Solenoid2=> O10B_ORING_LH_PUSHR_CYL_REV_FWD_Q1060_1, 
	AlarmSensor1=> OP10B_LH_PUSH_A1, 
	AlarmSensor2=> OP10B_LH_PUSH_A2, 
	AlarmSolenoid1=> OP10B_LH_PUSH_A3, 
	AlarmSolenoid2=> OP10B_LH_PUSH_A4, 
	AllSignal=> OP10B_LH_PUSH_A5, 
	AlarmPresent=> OP10B_CYLINDER_ERR.5, 
	Position1=> , 
	Position2=> , 
	HomeSensorBlink=> , 
	WorkSensorBlink=> ,
	Status:= OP10B_LH_PUSH_STUS,
	HMENG_RESULT := OP10B_HME_STP_NO);

// OP10B_LH_PUSH_CYLINDER_SAFE_WRK/HME
OP10B_RH_PUSH.SafeHome						:= OP10B_RH_GRP.Sensor2 ;
OP10B_RH_PUSH.SafeWork						:= OP10B_RH_GRP.Sensor2 ;

OP10B_RH_PUSH(
	Auto:= OP10B_AUTO_RUNNING OR OP10B_STEP_RUNNING OR OP10B_CYL_PNP_CHECK , 
	Manual:= OP10B_MANUAL_SELECTED,
	HOMING_RUNNING:= OP10B_START_HOMNG, 
	ErrorActive:= OP10B_ERR, 								(*OP10B_RH _ PUSHING CYL_FUNTIONAL_BLCK*)
	ResetPB:= Servo_Reset, 
	Sensor1:= NOT I10B_ORING_RH_PUSHR_CYL_REV_I1030_7, 
	Sensor2:=I10B_ORING_RH_PUSHR_CYL_REV_I1030_7 , 
	ManualPB1:=OP10B_MANUAL_SELECTED AND NOT OP10B_M_O_RHPUSH_CYL, 
	ManualPB2:=OP10B_MANUAL_SELECTED AND OP10B_M_O_RHPUSH_CYL, 
	AutoCmd1:=OP10B_RH_PUSH.Auto AND NOT OP10B_A_O_RHPUSH_CYL, 
	AutoCmd2:=OP10B_RH_PUSH.Auto AND OP10B_A_O_RHPUSH_CYL, 
	OperationEnable:= OperationEnable, 
	SafeHome:= 1, 
	SafeWork:= 1, 
	Pulse_1Sec:= Pulse_Block.Q1Hz, 
	BlinkingBit:= , 
	TimeOut1:= 5, 
	TimeOut2:= 5, 
	TimeOut3:= 5,
	HOMING_STRT:= (OP10B_HME_STP_NO=1),
	HME_DLY:= ,
	HME_DN_NO:= ,	
	HME_CYL_2:=TRUE ,
	HME_CYL_3:=TRUE , 
	Solenoid1=> , 
	Solenoid2=>O10B_ORING_RH_PUSHR_CYL_REV_FWD_Q1060_3 , 
	AlarmSensor1=> OP10B_RH_PUSH_A1, 
	AlarmSensor2=> OP10B_RH_PUSH_A2, 
	AlarmSolenoid1=> OP10B_RH_PUSH_A3, 
	AlarmSolenoid2=> OP10B_RH_PUSH_A4, 
	AllSignal=> OP10B_RH_PUSH_A5, 
	AlarmPresent=> OP10B_CYLINDER_ERR.6, 
	Position1=> , 
	Position2=> , 
	HomeSensorBlink=> , 
	WorkSensorBlink=> ,	
	Status:= OP10B_RH_PUSH_STUS,
	HMENG_RESULT := OP10B_PARLLEL);

// OP10B_LH_REJ_CYLINDER_SAFE_WRK/HME
//OP10B_LH_REJ.SafeHome						:= TRUE;
//OP10B_LH_REJ.SafeWork						:= TRUE;

OP10B_LH_REJ(
	Auto:= OP10B_AUTO_RUNNING OR OP10B_STEP_RUNNING OR OP10B_CYL_PNP_CHECK, 
	Manual:= OP10B_MANUAL_SELECTED,
	HOMING_RUNNING:= OP10B_START_HOMNG, 
	ErrorActive:= OP10B_ERR, 								(*OP10B_RH _ PUSHING CYL_FUNTIONAL_BLCK*)
	ResetPB:= Servo_Reset, 
	Sensor1:=I10B_LH_FIRTRE_ORING_REJ_CYL_REV_I1031_6, 											 
	Sensor2:=I10B_LH_FIRTRE_ORING_REJ_CYL_FWD_I1031_7,                                              
	ManualPB1:= OP10B_M_LH_REJ_HOME,                        
	ManualPB2:= OP10B_M_LH_REJ_WRK,
	AutoCmd1:= OP10B_A_LH_REJ_HOME,                                              
	AutoCmd2:= OP10B_A_LH_REJ_WRK,                                              
	OperationEnable:= OperationEnable, 
	SafeHome:= 1, 
	SafeWork:= 1, 
	Pulse_1Sec:= Pulse_Block.Q1Hz, 
	BlinkingBit:= , 
	TimeOut1:= 5, 
	TimeOut2:= 5, 
	TimeOut3:= 5,
	HOMING_STRT:= (OP10B_HME_STP_NO=1),
	HME_DLY:= ,
	HME_DN_NO:= ,
	HME_CYL_2:=TRUE ,
	HME_CYL_3:=TRUE , 
	Solenoid1=>O10B_LH_FIRTRE_ORING_REJ_CYL_REV_Q1061_2 , 
	Solenoid2=> O10B_LH_FIRTRE_ORING_REJ_CYL_FWD_Q1061_3, 
	AlarmSensor1=> OP10B_LH_REJ_A1,	
	AlarmSensor2=>OP10B_LH_REJ_A2,	
	AlarmSolenoid1=>OP10B_LH_REJ_A3,	
	AlarmSolenoid2=>OP10B_LH_REJ_A4,	
	AllSignal=> OP10B_LH_REJ_A5,	
	AlarmPresent=> OP10B_CYLINDER_ERR.7, 
	Position1=> , 
	Position2=> , 
	HomeSensorBlink=> , 
	WorkSensorBlink=> ,	
	Status:= OP10B_RH_PUSH_STUS,
	HMENG_RESULT := OP10B_PARLLEL);	
	
// OP10B_RH_REJ_CYLINDER_SAFE_WRK/HME
//OP10B_RH_REJ.SafeHome						:= TRUE;
//OP10B_RH_REJ.SafeWork						:= TRUE;

OP10B_RH_REJ(
	Auto:= OP10B_AUTO_RUNNING OR OP10B_STEP_RUNNING OR OP10B_CYL_PNP_CHECK, 
	Manual:= OP10B_MANUAL_SELECTED,
	HOMING_RUNNING:= OP10B_START_HOMNG, 
	ErrorActive:= OP10B_ERR, 								(*OP10B_RH _ PUSHING CYL_FUNTIONAL_BLCK*)
	ResetPB:= Servo_Reset, 
	Sensor1:= I10B_RH_FIRTRE_ORING_REJ_CYL_REV_I1040_0 , 
	Sensor2:= I10B_RH_FIRTRE_ORING_REJ_CYL_FWD_I1040_1 , 
	ManualPB1:= OP10B_M_RH_REJ_HOME,		
	ManualPB2:= OP10B_M_RH_REJ_WRK,	  
	AutoCmd1:= OP10B_A_RH_REJ_HOME, 
	AutoCmd2:= OP10B_A_RH_REJ_WRK, 
	OperationEnable:= OperationEnable, 
	SafeHome:= 1, 
	SafeWork:= 1, 
	Pulse_1Sec:= Pulse_Block.Q1Hz, 
	BlinkingBit:= , 
	TimeOut1:= 5, 
	TimeOut2:= 5, 
	TimeOut3:= 5,
	HOMING_STRT:= (OP10B_HME_STP_NO=1),
	HME_DLY:= ,
	HME_DN_NO:= ,
	HME_CYL_2:=TRUE ,
	HME_CYL_3:=TRUE , 
	Solenoid1=>O10B_RH_FIRTRE_ORING_REJ_CYL_REV_Q1061_4 , 
	Solenoid2=>O10B_RH_FIRTRE_ORING_REJ_CYL_FWD_Q1061_5 , 
	AlarmSensor1=> OP10B_RH_REJ_A1,	
	AlarmSensor2=> OP10B_RH_REJ_A2,	
	AlarmSolenoid1=> OP10B_RH_REJ_A3,	
	AlarmSolenoid2=>OP10B_RH_REJ_A4,	
	AllSignal=>OP10B_RH_REJ_A5,	
	AlarmPresent=> OP10B_CYLINDER_ERR.8, 
	Position1=> , 
	Position2=> , 
	HomeSensorBlink=> , 
	WorkSensorBlink=> ,	
	Status:= OP10B_RH_PUSH_STUS,
	HMENG_RESULT := OP10B_PARLLEL);	

	
////////////////////////////////////////OP10 SINGULATING GRIPPER/////////////////////////////


OP10_BDY_SING_FRT(
	Auto:= (OP10A_AUTO_RUNNING OR  OP10A_STEP_RUNNING )OR (OP10B_AUTO_RUNNING OR OP10B_STEP_RUNNING) OR CHECK, 
	Manual:= OP10B_MANUAL_SELECTED AND OP10A_MANUAL_SELECTED AND NOT CHECK,
	HOMING_RUNNING:= (OP10A_START_HOMNG OR OP10B_START_HOMNG), 
	ErrorActive:= (OP10B_ERR AND NOT OP10B_BYPASS) OR (OP10A_ERR AND NOT OP10A_BYPASS), 								(*OP10B_RH _ PUSHING CYL_FUNTIONAL_BLCK*)
	ResetPB:= Servo_Reset, 
	Sensor1:= I10A_BDY_SING_CYL_CLSE_I1020_2,  
	Sensor2:= I10A_BDY_SING_CYL_OPN_I1020_3,  
	ManualPB1:=OP10_FRT_BDY_SING_HME,											
	ManualPB2:=OP10_FRT_BDY_SING_WRK,	                                    	
	AutoCmd1:= OP10_A_FRT_BDY_SING_HME,                                        	
	AutoCmd2:= OP10_A_FRT_BDY_SING_WRK,                                        	
	OperationEnable:= OperationEnable, 
	SafeHome:= 1, 
	SafeWork:= 1, 
	Pulse_1Sec:= Pulse_Block.Q1Hz, 
	BlinkingBit:= , 
	TimeOut1:= 5, 
	TimeOut2:= 5, 
	TimeOut3:= 5,
	HOMING_STRT:= OP10_FRT_CYL_INITZAL,
	HME_DLY:= ,
	HME_DN_NO:= ,
	HME_CYL_2:=TRUE ,
	HME_CYL_3:=TRUE , 
	Solenoid1=>O10A_BDY_SING_CYL_CLSE_Q1051_6, 
	Solenoid2=>O10A_BDY_SING_CYL_OPN_Q1051_7,  
	AlarmSensor1=>OP10_BDY_SING_FRT_A1,	
	AlarmSensor2=>OP10_BDY_SING_FRT_A2,	
	AlarmSolenoid1=>OP10_BDY_SING_FRT_A3,	
	AlarmSolenoid2=>OP10_BDY_SING_FRT_A4,	
	AllSignal=>OP10_BDY_SING_FRT_A5,	
	AlarmPresent=> OP10A_CYLINDER_ERR.9, 
	Position1=> , 
	Position2=> , 
	HomeSensorBlink=> , 
	WorkSensorBlink=> ,	
	Status:= OP10_BDY_SING_FRT_STATUS,
	HMENG_RESULT := OP10B_PARLLEL);


OP10_BDY_SING_SEC(
	Auto:= (OP10A_AUTO_RUNNING OR  OP10A_STEP_RUNNING )OR (OP10B_AUTO_RUNNING OR OP10B_STEP_RUNNING) OR CHECK, 
	Manual:= OP10B_MANUAL_SELECTED AND OP10A_MANUAL_SELECTED AND NOT CHECK,
	HOMING_RUNNING:= (OP10A_START_HOMNG OR OP10B_START_HOMNG), 
	ErrorActive:= (OP10B_ERR AND NOT OP10B_BYPASS) OR (OP10A_ERR AND NOT OP10A_BYPASS), 								(*OP10B_RH _ PUSHING CYL_FUNTIONAL_BLCK*)
	ResetPB:= Servo_Reset, 
	Sensor1:= I10B_BDY_SING_CYL_CLSE_I1040_2,   
	Sensor2:= I10B_BDY_SING_CYL_OPN_I1040_3,   
	ManualPB1:=OP10_SEC_BDY_SING_HME,		
	ManualPB2:=OP10_SEC_BDY_SING_WRK,	  
	AutoCmd1:= OP10_A_SEC_BDY_SING_HME, 
	AutoCmd2:= OP10_A_SEC_BDY_SING_WRK, 
	OperationEnable:= OperationEnable, 
	SafeHome:= 1, 
	SafeWork:= 1, 
	Pulse_1Sec:= Pulse_Block.Q1Hz, 
	BlinkingBit:= , 
	TimeOut1:= 5, 
	TimeOut2:= 5, 
	TimeOut3:= 5,
	HOMING_STRT:=OP10_SEC_CYL_INITZAL,
	HME_DLY:= ,
	HME_DN_NO:= ,
	HME_CYL_2:=TRUE ,
	HME_CYL_3:=TRUE , 
	Solenoid1=> O10B_BDY_SING_CYL_CLSE_Q1061_6,  
	Solenoid2=> O10B_BDY_SING_CYL_OPN_Q1061_7,   
	AlarmSensor1=> , 
	AlarmSensor2=> , 
	AlarmSolenoid1=>, 
	AlarmSolenoid2=> , 
	AllSignal=> , 
	AlarmPresent=> OP10A_CYLINDER_ERR.10, 
	Position1=> , 
	Position2=> , 
	HomeSensorBlink=> , 
	WorkSensorBlink=> ,	
	HMENG_RESULT=>  , 
	Status:= OP10_BDY_SING_SEC_STATUS,
	HMENG_RESULT := OP10B_PARLLEL);

END_PROGRAM

// ---- POUs/Programs/OP10/OP10_SERVO.TcPOU
PROGRAM OP10_SERVO
VAR
// IN_RANGE
	OP10_BDY_GRP_FRT						: AXIS_REF;
	OP10_BDY_GRP_SEC						: AXIS_REF;	
	OP10A_LH_GRIPPER						: AXIS_REF;
	OP10A_RH_GRIPPER						: AXIS_REF;
	OP10A_LH_ROTARY							: AXIS_REF;
	OP10A_RH_ROTARY							: AXIS_REF;
	OP10A_CONVRY							: AXIS_REF;
	OP10B_LH_GRIPPER						: AXIS_REF;
	OP10B_RH_GRIPPER						: AXIS_REF;
	OP10B_LH_ROTARY							: AXIS_REF;
	OP10B_RH_ROTARY							: AXIS_REF;
	OP10B_CONVRY							: AXIS_REF;	
	OP10_SRV_BLCK_INTZ						: BOOL;
	FESTO_NOT_NEED							: BOOL;
	NOT_REQ									: BOOL;


OP10A_RH_GRP_TORQUE_APPLIED: LREAL;


	
	
	
	
END_VAR

VAR PERSISTENT
	OP10_SRV_FRT_BDYPCK_WRK_DEGREE			: LREAL;
	OP10_SRV_FRT_BDYPCK_HME_DEGREE			: LREAL;
	OP10_SRV_SCND_BDYPCK_WRK_DEGREE			: LREAL;
	OP10_SRV_SCND_BDYPCK_HME_DEGREE			: LREAL;

	OP10A_SRV_LH_GRP_HME_MM					: LREAL;
	OP10A_SRV_LH_GRP_WRK_MM					: LREAL;
	OP10A_SRV_RH_GRP_HME_MM					: LREAL;
	OP10A_SRV_RH_GRP_WRK_MM					: LREAL;
	OP10A_SRV_LH_BDYANG_HME_MM				: LREAL;
	OP10A_SRV_LH_BDYANG_CMR_MM				: LREAL;
	OP10A_SRV_LH_BDYANG_FITRE_MM			: LREAL;
	OP10A_SRV_LH_BDYANG_WRK_MM				: LREAL;
	OP10A_SRV_RH_BDYANG_HME_MM				: LREAL;
	OP10A_SRV_RH_BDYANG_CMR_MM				: LREAL;
	OP10A_SRV_RH_BDYANG_FITRE_MM			: LREAL;
	OP10A_SRV_RH_BDYANG_WRK_MM				: LREAL;

	OP10B_SRV_LH_WRK_MM						: LREAL;
	OP10B_SRV_LH_HME_MM						: LREAL;
	OP10B_SRV_RH_WRK_MM						: LREAL;
	OP10B_SRV_RH_HME_MM						: LREAL;
	OP10B_SRV_LH_BDYANG_HME_MM				: LREAL;
	OP10B_SRV_LH_BDYANG_CMR_MM				: LREAL;
	OP10B_SRV_LH_BDYANG_FITRE_MM			: LREAL;
	OP10B_SRV_LH_BDYANG_WRK_MM				: LREAL;
	OP10B_SRV_RH_BDYANG_HME_MM				: LREAL;
	OP10B_SRV_RH_BDYANG_CMR_MM				: LREAL;
	OP10B_SRV_RH_BDYANG_FITRE_MM			: LREAL;
	OP10B_SRV_RH_BDYANG_WRK_MM				: LREAL;	






	OP10A_LH_GRP_TORQUE_APPLIED				: LREAL;
END_VAR

////////////////////////OP10 BODY PICK ROTATE SERVO ///////////////////////////
IF OP10_A_SRV_FST_BDYPCK_WRK THEN
	OP10_SRV_FRST_PCKBDY_CNT.ABSmove_Start		:= TRUE;
	OP10_SRV_FRST_PCKBDY_CNT.Position			:= OP10_SRV_FRT_BDYPCK_WRK_DEGREE ;
IF OP10_SRV_FRST_PCKBDY_WRK_FB THEN
	OP10_SRV_FRST_PCKBDY_CNT.ABSmove_Start		:= FALSE;
	OP10_A_SRV_FST_BDYPCK_WRK                  	:= FALSE;
END_IF
END_IF

IF OP10_A_SRV_FST_BDYPCK_HME THEN
	OP10_SRV_FRST_PCKBDY_CNT.ABSmove_Start		:= TRUE;
	OP10_SRV_FRST_PCKBDY_CNT.Position			:= OP10_SRV_FRT_BDYPCK_HME_DEGREE ;
IF OP10_SRV_FRST_PCKBDY_HME_FB THEN
	OP10_SRV_FRST_PCKBDY_CNT.ABSmove_Start		:= FALSE;
	OP10_A_SRV_FST_BDYPCK_HME                  	:= FALSE;
END_IF
END_IF

IF OP10_A_SRV_SCND_BDYPCK_WRK THEN
	OP10_SRV_SCND_PCKBDY_CNT.ABSmove_Start		:= TRUE;
	OP10_SRV_SCND_PCKBDY_CNT.Position			:= OP10_SRV_SCND_BDYPCK_WRK_DEGREE ;
IF OP10_SRV_SCND_PCKBDY_WRK_FB THEN
	OP10_SRV_SCND_PCKBDY_CNT.ABSmove_Start		:= FALSE;
	OP10_A_SRV_SCND_BDYPCK_WRK                  := FALSE;
END_IF
END_IF

IF OP10_A_SRV_SCND_BDYPCK_HME THEN
	OP10_SRV_SCND_PCKBDY_CNT.ABSmove_Start		:= TRUE;
	OP10_SRV_SCND_PCKBDY_CNT.Position			:= OP10_SRV_SCND_BDYPCK_HME_DEGREE ;
IF OP10_SRV_SCND_PCKBDY_HME_FB THEN
	OP10_SRV_SCND_PCKBDY_CNT.ABSmove_Start		:= FALSE;
	OP10_A_SRV_SCND_BDYPCK_HME                 	:= FALSE;
END_IF
END_IF

///////////////////////////////////////////////////OP10A GRIPPER STEPPER/////////////////////////////////////////////

IF OP10A_A_SRV_LH_GRPWRK THEN
	OP10A_SRV_LH_BDYGRP_CNT.ABSmove_Start		:= TRUE;
	OP10A_SRV_LH_BDYGRP_CNT.Position			:= OP10A_SRV_LH_GRP_WRK_MM;
IF OP10A_A_SRV_LH_GRPWRK_FB THEN
	OP10A_A_SRV_LH_GRPWRK						:= FALSE;
	OP10A_SRV_LH_BDYGRP_CNT.ABSmove_Start		:= FALSE;		
END_IF
END_IF

IF OP10A_A_SRV_LH_GRPHME THEN
	OP10A_SRV_LH_BDYGRP_CNT.ABSmove_Start		:= TRUE;
	OP10A_SRV_LH_BDYGRP_CNT.Position			:= OP10A_SRV_LH_GRP_HME_MM;
IF OP10A_A_SRV_LH_GRPHME_FB THEN
	OP10A_A_SRV_LH_GRPHME						:= FALSE;
	OP10A_SRV_LH_BDYGRP_CNT.ABSmove_Start		:= FALSE;		
END_IF
END_IF

IF OP10A_A_SRV_RH_GRPWRK THEN
	OP10A_SRV_RH_BDYGRP_CNT.ABSmove_Start		:= TRUE;
	OP10A_SRV_RH_BDYGRP_CNT.Position			:= OP10A_SRV_RH_GRP_WRK_MM;
IF OP10A_A_SRV_RH_GRPWRK_FB THEN
	OP10A_A_SRV_RH_GRPWRK						:= FALSE;
	OP10A_SRV_RH_BDYGRP_CNT.ABSmove_Start		:= FALSE;		
END_IF
END_IF

IF OP10A_A_SRV_RH_GRPHME THEN
	OP10A_SRV_RH_BDYGRP_CNT.ABSmove_Start		:= TRUE;
	OP10A_SRV_RH_BDYGRP_CNT.Position			:= OP10A_SRV_RH_GRP_HME_MM;
IF OP10A_A_SRV_RH_GRPHME_FB THEN
	OP10A_A_SRV_RH_GRPHME						:= FALSE;
	OP10A_SRV_RH_BDYGRP_CNT.ABSmove_Start		:= FALSE;		
END_IF
END_IF

//////////////////////////////////////OP10A ANGLE ROTATE /////////////////////

IF OP10A_SRV_LH_BDYANG_HME THEN
	OP10A_SRV_LH_BDYANG_CNT.ABSmove_Start		:= TRUE;
	OP10A_SRV_LH_BDYANG_CNT.Position			:= OP10A_SRV_LH_BDYANG_HME_MM;
IF OP10A_SRV_LH_BDYANG_HME_FB THEN
	OP10A_SRV_LH_BDYANG_HME						:= FALSE;
	OP10A_SRV_LH_BDYANG_CNT.ABSmove_Start		:= FALSE;	
END_IF
END_IF

IF OP10A_SRV_LH_BDYANG_CMR THEN
	OP10A_SRV_LH_BDYANG_CNT.ABSmove_Start		:= TRUE;
	OP10A_SRV_LH_BDYANG_CNT.Position			:= OP10A_SRV_LH_BDYANG_CMR_MM;
IF OP10A_SRV_LH_BDYANG_CMR_FB THEN
	OP10A_SRV_LH_BDYANG_CMR						:= FALSE;
	OP10A_SRV_LH_BDYANG_CNT.ABSmove_Start		:= FALSE;	
END_IF
END_IF

IF OP10A_SRV_LH_BDYANG_FITRE THEN
	OP10A_SRV_LH_BDYANG_CNT.ABSmove_Start		:= TRUE;
	OP10A_SRV_LH_BDYANG_CNT.Position			:= OP10A_SRV_LH_BDYANG_FITRE_MM;
IF OP10A_SRV_LH_BDYANG_FITRE_FB THEN
	OP10A_SRV_LH_BDYANG_FITRE					:= FALSE;
	OP10A_SRV_LH_BDYANG_CNT.ABSmove_Start		:= FALSE;	
END_IF
END_IF

IF OP10A_SRV_LH_BDYANG_WRK THEN
	OP10A_SRV_LH_BDYANG_CNT.ABSmove_Start		:= TRUE;
	OP10A_SRV_LH_BDYANG_CNT.Position			:= OP10A_SRV_LH_BDYANG_WRK_MM;
IF OP10A_SRV_LH_BDYANG_WRK_FB THEN
	OP10A_SRV_LH_BDYANG_WRK						:= FALSE;
	OP10A_SRV_LH_BDYANG_CNT.ABSmove_Start		:= FALSE;	
END_IF
END_IF

IF OP10A_SRV_RH_BDYANG_HME THEN
	OP10A_SRV_RH_BDYANG_CNT.ABSmove_Start		:= TRUE;
	OP10A_SRV_RH_BDYANG_CNT.Position			:= OP10A_SRV_RH_BDYANG_HME_MM;
IF OP10A_SRV_RH_BDYANG_HME_FB THEN
	OP10A_SRV_RH_BDYANG_HME						:= FALSE;
	OP10A_SRV_RH_BDYANG_CNT.ABSmove_Start		:= FALSE;	
END_IF
END_IF

IF OP10A_SRV_RH_BDYANG_CMR THEN
	OP10A_SRV_RH_BDYANG_CNT.ABSmove_Start		:= TRUE;
	OP10A_SRV_RH_BDYANG_CNT.Position			:= OP10A_SRV_RH_BDYANG_CMR_MM;
IF OP10A_SRV_RH_BDYANG_CMR_FB THEN
	OP10A_SRV_RH_BDYANG_CMR						:= FALSE;
	OP10A_SRV_RH_BDYANG_CNT.ABSmove_Start		:= FALSE;	
END_IF
END_IF

IF OP10A_SRV_RH_BDYANG_FITRE THEN
	OP10A_SRV_RH_BDYANG_CNT.ABSmove_Start		:= TRUE;
	OP10A_SRV_RH_BDYANG_CNT.Position			:= OP10A_SRV_RH_BDYANG_FITRE_MM;
IF OP10A_SRV_RH_BDYANG_FITRE_FB THEN
	OP10A_SRV_RH_BDYANG_FITRE					:= FALSE;
	OP10A_SRV_RH_BDYANG_CNT.ABSmove_Start		:= FALSE;	
END_IF
END_IF

IF OP10A_SRV_RH_BDYANG_WRK THEN
	OP10A_SRV_RH_BDYANG_CNT.ABSmove_Start		:= TRUE;
	OP10A_SRV_RH_BDYANG_CNT.Position			:= OP10A_SRV_RH_BDYANG_WRK_MM;
IF OP10A_SRV_LH_BDYANG_WRK_FB THEN
	OP10A_SRV_RH_BDYANG_WRK						:= FALSE;
	OP10A_SRV_RH_BDYANG_CNT.ABSmove_Start		:= FALSE;	
END_IF
END_IF

/////////////////////////////////////////////////////OP10B ////////////////////////////////////////////////////

IF OP10B_A_SRV_LH_GRPWRK THEN
	OP10B_SRV_LH_BDYGRP_CNT.ABSmove_Start		:= TRUE;
	OP10B_SRV_LH_BDYGRP_CNT.Position			:= OP10B_SRV_LH_WRK_MM;
IF OP10B_A_SRV_LH_GRPWRK_FB THEN
	OP10B_A_SRV_LH_GRPWRK						:= FALSE;
	OP10B_SRV_LH_BDYGRP_CNT.ABSmove_Start		:= FALSE;		
END_IF
END_IF

IF OP10B_A_SRV_LH_GRPHME THEN
	OP10B_SRV_LH_BDYGRP_CNT.ABSmove_Start		:= TRUE;
	OP10B_SRV_LH_BDYGRP_CNT.Position			:= OP10B_SRV_LH_HME_MM;
IF OP10B_A_SRV_LH_GRPHME_FB THEN
	OP10B_A_SRV_LH_GRPHME						:= FALSE;
	OP10B_SRV_LH_BDYGRP_CNT.ABSmove_Start		:= FALSE;		
END_IF
END_IF

IF OP10B_A_SRV_RH_GRPWRK THEN
	OP10B_SRV_RH_BDYGRP_CNT.ABSmove_Start		:= TRUE;
	OP10B_SRV_RH_BDYGRP_CNT.Position			:= OP10B_SRV_RH_WRK_MM;
IF OP10B_A_SRV_RH_GRPWRK_FB THEN
	OP10B_A_SRV_RH_GRPWRK						:= FALSE;
	OP10B_SRV_RH_BDYGRP_CNT.ABSmove_Start		:= FALSE;		
END_IF
END_IF

IF OP10B_A_SRV_RH_GRPHME THEN
	OP10B_SRV_RH_BDYGRP_CNT.ABSmove_Start		:= TRUE;
	OP10B_SRV_RH_BDYGRP_CNT.Position			:= OP10B_SRV_RH_HME_MM;
IF OP10B_A_SRV_RH_GRPHME_FB THEN
	OP10B_A_SRV_RH_GRPHME						:= FALSE;
	OP10B_SRV_RH_BDYGRP_CNT.ABSmove_Start		:= FALSE;		
END_IF
END_IF

//////////////////////////////////////OP10B ANGLE ROTATE /////////////////////

IF OP10B_SRV_LH_BDYANG_HME THEN
	OP10B_SRV_LH_BDYANG_CNT.ABSmove_Start		:= TRUE;
	OP10B_SRV_LH_BDYANG_CNT.Position			:= OP10B_SRV_LH_BDYANG_HME_MM;
IF OP10B_SRV_LH_BDYANG_HME_FB THEN
	OP10B_SRV_LH_BDYANG_HME						:= FALSE;
	OP10B_SRV_LH_BDYANG_CNT.ABSmove_Start		:= FALSE;	
END_IF
END_IF


IF OP10B_SRV_LH_BDYANG_CMR THEN
	OP10B_SRV_LH_BDYANG_CNT.ABSmove_Start		:= TRUE;
	OP10B_SRV_LH_BDYANG_CNT.Position			:= OP10B_SRV_LH_BDYANG_CMR_MM;
IF OP10B_SRV_LH_BDYANG_CMR_FB THEN
	OP10B_SRV_LH_BDYANG_CMR						:= FALSE;
	OP10B_SRV_LH_BDYANG_CNT.ABSmove_Start		:= FALSE;	
END_IF
END_IF

IF OP10B_SRV_LH_BDYANG_FITRE THEN
	OP10B_SRV_LH_BDYANG_CNT.ABSmove_Start		:= TRUE;
	OP10B_SRV_LH_BDYANG_CNT.Position			:= OP10B_SRV_LH_BDYANG_FITRE_MM;
IF OP10B_SRV_LH_BDYANG_FITRE_FB THEN
	OP10B_SRV_LH_BDYANG_FITRE					:= FALSE;
	OP10B_SRV_LH_BDYANG_CNT.ABSmove_Start		:= FALSE;	
END_IF
END_IF

IF OP10B_SRV_LH_BDYANG_WRK THEN
	OP10B_SRV_LH_BDYANG_CNT.ABSmove_Start		:= TRUE;
	OP10B_SRV_LH_BDYANG_CNT.Position			:= OP10B_SRV_LH_BDYANG_WRK_MM;
IF OP10B_SRV_LH_BDYANG_WRK_FB THEN
	OP10B_SRV_LH_BDYANG_WRK						:= FALSE;
	OP10B_SRV_LH_BDYANG_CNT.ABSmove_Start		:= FALSE;	
END_IF
END_IF

IF OP10B_SRV_RH_BDYANG_HME THEN
	OP10B_SRV_RH_BDYANG_CNT.ABSmove_Start		:= TRUE;
	OP10B_SRV_RH_BDYANG_CNT.Position			:= OP10B_SRV_RH_BDYANG_HME_MM;
IF OP10B_SRV_RH_BDYANG_HME_FB THEN
	OP10B_SRV_RH_BDYANG_HME						:= FALSE;
	OP10B_SRV_RH_BDYANG_CNT.ABSmove_Start		:= FALSE;	
END_IF
END_IF

IF OP10B_SRV_RH_BDYANG_CMR THEN
	OP10B_SRV_RH_BDYANG_CNT.ABSmove_Start		:= TRUE;
	OP10B_SRV_RH_BDYANG_CNT.Position			:= OP10B_SRV_RH_BDYANG_CMR_MM;
IF OP10B_SRV_RH_BDYANG_CMR_FB THEN
	OP10B_SRV_RH_BDYANG_CMR						:= FALSE;
	OP10B_SRV_RH_BDYANG_CNT.ABSmove_Start		:= FALSE;	
END_IF
END_IF

IF OP10B_SRV_RH_BDYANG_FITRE THEN
	OP10B_SRV_RH_BDYANG_CNT.ABSmove_Start		:= TRUE;
	OP10B_SRV_RH_BDYANG_CNT.Position			:= OP10B_SRV_RH_BDYANG_FITRE_MM;
IF OP10B_SRV_RH_BDYANG_FITRE_FB THEN
	OP10B_SRV_RH_BDYANG_FITRE					:= FALSE;
	OP10B_SRV_RH_BDYANG_CNT.ABSmove_Start		:= FALSE;	
END_IF
END_IF

IF OP10B_SRV_RH_BDYANG_WRK THEN
	OP10B_SRV_RH_BDYANG_CNT.ABSmove_Start		:= TRUE;
	OP10B_SRV_RH_BDYANG_CNT.Position			:= OP10B_SRV_RH_BDYANG_WRK_MM;
IF OP10B_SRV_RH_BDYANG_WRK_FB THEN
	OP10B_SRV_RH_BDYANG_WRK						:= FALSE;
	OP10B_SRV_RH_BDYANG_CNT.ABSmove_Start		:= FALSE;	
END_IF
END_IF



// SERVO_POSITION_STATUS
								(*OP10*)
	OP10_SRV_FRST_PCKBDY_WRK_FB					:= OP10_SRV_FRST_PCKBDY_CNT.Axis_In_Pos AND In_Range(value:=OP10_SRV_FRST_PCKBDY_STUS.actualPosition , setvalue:=OP10_SRV_FRT_BDYPCK_WRK_DEGREE , tolerance:=0.1);
	OP10_SRV_FRST_PCKBDY_HME_FB					:= OP10_SRV_FRST_PCKBDY_CNT.Axis_In_Pos AND In_Range(value:=OP10_SRV_FRST_PCKBDY_STUS.actualPosition , setvalue:=OP10_SRV_FRT_BDYPCK_HME_DEGREE , tolerance:=0.1);
	OP10_SRV_SCND_PCKBDY_WRK_FB					:= OP10_SRV_SCND_PCKBDY_CNT.Axis_In_Pos AND In_Range(value:=OP10_SRV_SCND_PCKBDY_STUS.actualPosition , setvalue:=OP10_SRV_SCND_BDYPCK_WRK_DEGREE , tolerance:=0.1);
	OP10_SRV_SCND_PCKBDY_HME_FB					:= OP10_SRV_SCND_PCKBDY_CNT.Axis_In_Pos AND In_Range(value:=OP10_SRV_SCND_PCKBDY_STUS.actualPosition , setvalue:=OP10_SRV_SCND_BDYPCK_HME_DEGREE , tolerance:=0.1);
								(*OP10A*)
	OP10A_A_SRV_LH_GRPWRK_FB					:= OP10A_SRV_LH_BDYGRP_CNT.Axis_In_Pos AND In_Range(value:=OP10A_SRV_LH_BDYGRP_STUS.actualPosition , setvalue:=OP10A_SRV_LH_GRP_WRK_MM , tolerance:=0.5);
	OP10A_A_SRV_LH_GRPHME_FB					:= OP10A_SRV_LH_BDYGRP_CNT.Axis_In_Pos AND In_Range(value:=OP10A_SRV_LH_BDYGRP_STUS.actualPosition , setvalue:=OP10A_SRV_LH_GRP_HME_MM , tolerance:=0.5);
	OP10A_A_SRV_RH_GRPWRK_FB					:= OP10A_SRV_RH_BDYGRP_CNT.Axis_In_Pos AND In_Range(value:=OP10A_SRV_RH_BDYGRP_STUS.actualPosition , setvalue:=OP10A_SRV_RH_GRP_WRK_MM , tolerance:=0.5);
	OP10A_A_SRV_RH_GRPHME_FB					:= OP10A_SRV_RH_BDYGRP_CNT.Axis_In_Pos AND In_Range(value:=OP10A_SRV_RH_BDYGRP_STUS.actualPosition , setvalue:=OP10A_SRV_RH_GRP_HME_MM , tolerance:=0.5);
	OP10A_SRV_LH_BDYANG_HME_FB					:= OP10A_SRV_LH_BDYANG_CNT.Axis_In_Pos AND In_Range(value:=OP10A_SRV_LH_BDYANG_STUS.actualPosition , setvalue:=OP10A_SRV_LH_BDYANG_HME_MM , tolerance:=1);
	OP10A_SRV_LH_BDYANG_WRK_FB					:= OP10A_SRV_LH_BDYANG_CNT.Axis_In_Pos AND In_Range(value:=OP10A_SRV_LH_BDYANG_STUS.actualPosition , setvalue:=OP10A_SRV_LH_BDYANG_WRK_MM , tolerance:=1);
	OP10A_SRV_RH_BDYANG_HME_FB					:= OP10A_SRV_RH_BDYANG_CNT.Axis_In_Pos AND In_Range(value:=OP10A_SRV_RH_BDYANG_STUS.actualPosition , setvalue:=OP10A_SRV_RH_BDYANG_HME_MM , tolerance:=1);
	OP10A_SRV_RH_BDYANG_WRK_FB                  := OP10A_SRV_RH_BDYANG_CNT.Axis_In_Pos AND In_Range(value:=OP10A_SRV_RH_BDYANG_STUS.actualPosition , setvalue:=OP10A_SRV_RH_BDYANG_WRK_MM , tolerance:=1);
	OP10A_SRV_LH_BDYANG_ZERO_FB					:= OP10A_SRV_LH_BDYANG_CNT.Axis_In_Pos AND In_Range(value:=OP10A_SRV_LH_BDYANG_STUS.actualPosition , setvalue:=0 , tolerance:=1);
	OP10A_SRV_RH_BDYANG_ZERO_FB                 := OP10A_SRV_RH_BDYANG_CNT.Axis_In_Pos AND In_Range(value:=OP10A_SRV_RH_BDYANG_STUS.actualPosition , setvalue:=0 , tolerance:=1);
	OP10A_SRV_LH_BDYANG_CMR_FB					:= OP10A_SRV_LH_BDYANG_CNT.Axis_In_Pos AND In_Range(value:=OP10A_SRV_LH_BDYANG_STUS.actualPosition , setvalue:=OP10A_SRV_LH_BDYANG_CMR_MM , tolerance:=1);
    OP10A_SRV_LH_BDYANG_FITRE_FB	            := OP10A_SRV_LH_BDYANG_CNT.Axis_In_Pos AND In_Range(value:=OP10A_SRV_LH_BDYANG_STUS.actualPosition , setvalue:=OP10A_SRV_LH_BDYANG_FITRE_MM , tolerance:=1);
	OP10A_SRV_RH_BDYANG_CMR_FB		            := OP10A_SRV_RH_BDYANG_CNT.Axis_In_Pos AND In_Range(value:=OP10A_SRV_RH_BDYANG_STUS.actualPosition , setvalue:=OP10A_SRV_RH_BDYANG_CMR_MM , tolerance:=1);
    OP10A_SRV_RH_BDYANG_FITRE_FB	            := OP10A_SRV_RH_BDYANG_CNT.Axis_In_Pos AND In_Range(value:=OP10A_SRV_RH_BDYANG_STUS.actualPosition , setvalue:=OP10A_SRV_RH_BDYANG_FITRE_MM , tolerance:=1);
								(*OP10B*)
	OP10B_A_SRV_LH_GRPWRK_FB					:= OP10B_SRV_LH_BDYGRP_CNT.Axis_In_Pos AND In_Range(value:=OP10B_SRV_LH_BDYGRP_STUS.actualPosition , setvalue:=OP10B_SRV_LH_WRK_MM , tolerance:=0.5);
	OP10B_A_SRV_LH_GRPHME_FB					:= OP10B_SRV_LH_BDYGRP_CNT.Axis_In_Pos AND In_Range(value:=OP10B_SRV_LH_BDYGRP_STUS.actualPosition , setvalue:=OP10B_SRV_LH_HME_MM , tolerance:=0.5);
	OP10B_A_SRV_RH_GRPWRK_FB					:= OP10B_SRV_RH_BDYGRP_CNT.Axis_In_Pos AND In_Range(value:=OP10B_SRV_RH_BDYGRP_STUS.actualPosition , setvalue:=OP10B_SRV_RH_WRK_MM , tolerance:=0.5);
	OP10B_A_SRV_RH_GRPHME_FB					:= OP10B_SRV_RH_BDYGRP_CNT.Axis_In_Pos AND In_Range(value:=OP10B_SRV_RH_BDYGRP_STUS.actualPosition , setvalue:=OP10B_SRV_RH_HME_MM , tolerance:=0.5);
	OP10B_SRV_LH_BDYANG_HME_FB					:= OP10B_SRV_LH_BDYANG_CNT.Axis_In_Pos AND In_Range(value:=OP10B_SRV_LH_BDYANG_STUS.actualPosition , setvalue:=OP10B_SRV_LH_BDYANG_HME_MM , tolerance:=1);
	OP10B_SRV_LH_BDYANG_WRK_FB					:= OP10B_SRV_LH_BDYANG_CNT.Axis_In_Pos AND In_Range(value:=OP10B_SRV_LH_BDYANG_STUS.actualPosition , setvalue:=OP10B_SRV_LH_BDYANG_WRK_MM , tolerance:=1);
	OP10B_SRV_RH_BDYANG_HME_FB					:= OP10B_SRV_RH_BDYANG_CNT.Axis_In_Pos AND In_Range(value:=OP10B_SRV_RH_BDYANG_STUS.actualPosition , setvalue:=OP10B_SRV_RH_BDYANG_HME_MM , tolerance:=1);
	OP10B_SRV_RH_BDYANG_WRK_FB                  := OP10B_SRV_RH_BDYANG_CNT.Axis_In_Pos AND In_Range(value:=OP10B_SRV_RH_BDYANG_STUS.actualPosition , setvalue:=OP10B_SRV_RH_BDYANG_WRK_MM , tolerance:=1);
	OP10B_SRV_LH_BDYANG_ZERO_FB					:= OP10B_SRV_LH_BDYANG_CNT.Axis_In_Pos AND In_Range(value:=OP10B_SRV_LH_BDYANG_STUS.actualPosition , setvalue:=0 , tolerance:=1);
	OP10B_SRV_RH_BDYANG_ZERO_FB                 := OP10B_SRV_RH_BDYANG_CNT.Axis_In_Pos  AND In_Range(value:=OP10B_SRV_RH_BDYANG_STUS.actualPosition , setvalue:=0 , tolerance:=1);
	OP10B_SRV_LH_BDYANG_CMR_FB					:= OP10B_SRV_LH_BDYANG_CNT.Axis_In_Pos AND In_Range(value:=OP10B_SRV_LH_BDYANG_STUS.actualPosition , setvalue:=OP10B_SRV_LH_BDYANG_CMR_MM , tolerance:=1);
    OP10B_SRV_LH_BDYANG_FITRE_FB	            := OP10B_SRV_LH_BDYANG_CNT.Axis_In_Pos AND In_Range(value:=OP10B_SRV_LH_BDYANG_STUS.actualPosition , setvalue:=OP10B_SRV_LH_BDYANG_FITRE_MM , tolerance:=1);
	OP10B_SRV_RH_BDYANG_CMR_FB		            := OP10B_SRV_RH_BDYANG_CNT.Axis_In_Pos AND In_Range(value:=OP10B_SRV_RH_BDYANG_STUS.actualPosition , setvalue:=OP10B_SRV_RH_BDYANG_CMR_MM , tolerance:=1);
    OP10B_SRV_RH_BDYANG_FITRE_FB	            := OP10B_SRV_RH_BDYANG_CNT.Axis_In_Pos AND In_Range(value:=OP10B_SRV_RH_BDYANG_STUS.actualPosition , setvalue:=OP10B_SRV_RH_BDYANG_FITRE_MM , tolerance:=1);
	
	
///////////////////////////ALL SERVO IN HOME////////////////////////////////////////	
	
IF OP10_SRV_FRST_PCKBDY_HME_FB AND OP10_SRV_SCND_PCKBDY_HME_FB  THEN
	OP10_SRV_ALL_HOME							:= TRUE;
ELSE
	OP10_SRV_ALL_HOME							:= FALSE;	
END_IF
	
IF OP10A_A_SRV_LH_GRPHME_FB AND OP10A_A_SRV_RH_GRPHME_FB AND OP10A_SRV_LH_BDYANG_HME_FB AND OP10A_SRV_RH_BDYANG_HME_FB  THEN
	OP10A_SRV_ALL_HOME							:= TRUE;
ELSE
	OP10A_SRV_ALL_HOME							:= FALSE;
END_IF
	
IF OP10B_A_SRV_LH_GRPHME_FB AND OP10B_A_SRV_RH_GRPHME_FB AND OP10B_SRV_LH_BDYANG_HME_FB AND OP10B_SRV_RH_BDYANG_HME_FB  THEN
	OP10B_SRV_ALL_HOME							:= TRUE;
ELSE
	OP10B_SRV_ALL_HOME							:= FALSE;
END_IF
	
OP10_FRT_BDY_GPR(
	bAxis1_Ref_Switch:= , 																// NOT USED 
	bInit:= OP10_SRV_BLCK_INTZ, 														// INITIALIZE ALL MC_BLOCK
	bErrorReset:= Servo_Reset , 														// ERROR RESET
	bEnable:= Servo_Enable,																// MC_POWER ON
	bMoveVelocity:= ,																	// MC_MOVE_VELOCITY_BLOCK 
	bHalt:= ,																			// MC_HALT 
	bManualMode:= OP10A_MANUAL_SELECTED AND OP10B_MANUAL_SELECTED, 														// MANUAL MODE SELECTED
	fHomePos:= , 																		// SET CURRENT POSSION AS GIVEN VALUE 
	fOverride:= , 																		// OVERRIDE_ALWAYS_100
	fTargetPosition:= OP10_SRV_FRST_PCKBDY_CNT.Position,								// TARGET POSITION DURING AUTO LOGIC 
	fTargetVelocity:= OP10_SERVO_POS_VEL_LIMIT.OP10_FIRST_BODY_VELOCITY, 																// TARGET VELOCITY DURING AUTO LOGIC
	fAcc:= , 																			// ACCLERATION DURING AUTO
	fDec:= ,																			// DEC DURING AUTO 
	Servo_High_Limit:= OP10_SERVO_POS_VEL_LIMIT.OP10_FIRST_BODY_PIC_POS_LIMIT,																	
	Servo_Low_Limit:=OP10_SERVO_POS_VEL_LIMIT.OP10_FIRST_BODY_PIC_NEG_LIMIT,	 	
	WARNING_LIMIT:=1, 																			
	Safe_move_Conditions:=Servo_Safety,
	TORQUE_APPLIED := ,													// SAFE TO MOVE OR OVERRIDE IS DISABLED 
	Axis:= OP10_BDY_GRP_FRT,															// AXIS REFERENCE 
	bHome:= OP10_SRV_FRST_PCKBDY_CNT.Axis_Home_Cmd, 									// START HOMING TO HOMING BLOCK								
	bSetPosition:= FESTO_NOT_NEED ,														// SET CURRENT POSITION AS HOME
	bMoveAbsolute:= OP10_SRV_FRST_PCKBDY_CNT.ABSmove_Start,								// START ABS MOVE
	bMoveRelative:= NOT_REQ , 															// START RELATIVE
	bMoveTorque:= NOT_REQ ,																// START TORQUE 
	stManualModeAxis:= OP10_SRV_FRST_PCKBDY_STUS, 										// MANUAL MODE CONTROL FOR JOG 	
	sAxisState=> OP10_SRV_FRST_PCKBDY_CNT.Axis_State,                                      								
	bAxis_ready=> , 																	// SERVO READY
	bAxisInPosition=> , 																
	bAxisError=> OP10_SRV_FRST_PCKBDY_CNT.Axis_Error, 																		// SERVO IN ERROR
	bAxisEnabled=> ,																	// SERVO ENABLED 
	bAxisHomed=> , 																		// SERVO  REACHED HOME FROM FUNTIONAL BLOCK
	bSetPositionDone=> ,                                								
	bHaltDone=> , 																		// SERVO HALT D0NE
	bSTOPDone=> , 																		// STOPED DURING ERR
	bHomeDone=> OP10_SRV_FRST_PCKBDY_CNT.Axis_In_Home, 																		// HOMING DONE FB
	bDone=> ,
	bTorqueReached=> ,                                  								
	bsafe_to_move=> , 																	// SAFE TO MOVE CONDITION FB
	baxis_in_home_pos=> , 																// SERVO ON HOME POSITION THROUGH CALCULATION
	bABS_Pos_done=> OP10_SRV_FRST_PCKBDY_CNT.Axis_In_Pos, 								// SERVO IN POSITION
	Actual_position=>OP10_SRV_FRST_PCKBDY_CNT.Actual_Position,																// ACTUAL POSITION
	Actual_velocity=> , 																// ACTUAL VELOCITY
	Actual_Torque=> );																	// ACTUAL TORQUE
	
OP10_SEC_BDY_GPR(
	bAxis1_Ref_Switch:= , 
	bInit:= OP10_SRV_BLCK_INTZ , 
	bErrorReset:= Servo_Reset , 
	bEnable:= Servo_Enable, 
	bMoveVelocity:= , 
	bHalt:= , 
	bManualMode:= OP10A_MANUAL_SELECTED AND OP10B_MANUAL_SELECTED, 
	fHomePos:= , 
	fOverride:= , 
	fTargetPosition:= OP10_SRV_SCND_PCKBDY_CNT.Position, 
	fTargetVelocity:= OP10_SERVO_POS_VEL_LIMIT.OP10_SECOND_BODY_VELOCITY, 
	fAcc:= , 
	fDec:= ,
	Servo_High_Limit:= OP10_SERVO_POS_VEL_LIMIT.OP10_SECOND_BODY_PIC_POS_LIMIT,																	
	Servo_Low_Limit:=OP10_SERVO_POS_VEL_LIMIT.OP10_SECOND_BODY_PIC_NEG_LIMIT,	 	
	WARNING_LIMIT:=1, 
	Safe_move_Conditions:= Servo_Safety,
	TORQUE_APPLIED := , 
	Axis:= OP10_BDY_GRP_SEC, 
	bHome:= OP10_SRV_SCND_PCKBDY_CNT.Axis_Home_Cmd, 
	bSetPosition:= FESTO_NOT_NEED , 
	bMoveAbsolute:= OP10_SRV_SCND_PCKBDY_CNT.ABSmove_Start, 
	bMoveRelative:= NOT_REQ , 
	bMoveTorque:= NOT_REQ , 
	stManualModeAxis:= OP10_SRV_SCND_PCKBDY_STUS,
	sAxisState=>OP10_SRV_SCND_PCKBDY_CNT.Axis_State , 
	bAxis_ready=> , 
	bAxisInPosition=> , 
	bAxisError=> OP10_SRV_SCND_PCKBDY_CNT.Axis_Error, 
	bAxisEnabled=> , 
	bAxisHomed=> , 
	bSetPositionDone=> , 
	bHaltDone=> , 
	bSTOPDone=> , 
	bHomeDone=> OP10_SRV_SCND_PCKBDY_CNT.Axis_In_Home, 
	bDone=> , 
	bTorqueReached=> , 
	bsafe_to_move=> , 
	baxis_in_home_pos=> , 
	bABS_Pos_done=> OP10_SRV_SCND_PCKBDY_CNT.Axis_In_Pos, 
	Actual_position=>OP10_SRV_SCND_PCKBDY_CNT.Actual_Position, 
	Actual_velocity=> , 
	Actual_Torque=> );


///////////////////////////////////		OP10A	///////////////////////////////


	
OP10A_LH_ROTY(
	bAxis1_Ref_Switch:= , 
	bInit:= OP10_SRV_BLCK_INTZ , 
	bErrorReset:= Servo_Reset, 
	bEnable:= Servo_Enable  , 
	bMoveVelocity:= , 
	bHalt:= , 
	bManualMode:= OP10A_MANUAL_SELECTED , 
	fHomePos:= , 
	fOverride:= , 
	fTargetPosition:= OP10A_SRV_LH_BDYANG_CNT.Position, 
	fTargetVelocity:= OP10_SERVO_POS_VEL_LIMIT.OP10A_LH_ROTRY_VELOCITY, 
	fAcc:= , 
	fDec:= ,
	Servo_High_Limit:= OP10_SERVO_POS_VEL_LIMIT.OP10A_LH_ROTRY_POS_LIMIT,																	
	Servo_Low_Limit:=OP10_SERVO_POS_VEL_LIMIT.OP10A_LH_GRPR_NEG_LIMIT, 
	Safe_move_Conditions:=Servo_Safety,
	TORQUE_APPLIED := , 
	Axis:= OP10A_LH_ROTARY, 
	bHome:= OP10A_SRV_LH_BDYANG_CNT.Axis_Home_Cmd, 
	bSetPosition:= FESTO_NOT_NEED , 
	bMoveAbsolute:= OP10A_SRV_LH_BDYANG_CNT.ABSmove_Start, 
	bMoveRelative:= NOT_REQ , 
	bMoveTorque:= NOT_REQ , 
	stManualModeAxis:= OP10A_SRV_LH_BDYANG_STUS, 
 	sAxisState=> OP10A_SRV_LH_BDYANG_CNT.Axis_State, 
	bAxis_ready=> , 
	bAxisInPosition=> , 
	bAxisError=> OP10A_SRV_LH_BDYANG_CNT.Axis_Error, 
	bAxisEnabled=> , 
	bAxisHomed=> , 
	bSetPositionDone=> , 
	bHaltDone=> , 
	bSTOPDone=> , 
	bHomeDone=> OP10A_SRV_LH_BDYANG_CNT.Axis_In_Home, 
	bDone=> , 
	bTorqueReached=> , 
	bsafe_to_move=> , 
	baxis_in_home_pos=> , 
	bABS_Pos_done=> OP10A_SRV_LH_BDYANG_CNT.Axis_In_Pos, 
	Actual_position=>,
	Actual_velocity=> , 
	Actual_Torque=> );
	
OP10A_RH_ROTY(
	bAxis1_Ref_Switch:= , 
	bInit:= OP10_SRV_BLCK_INTZ , 
	bErrorReset:= Servo_Reset, 
	bEnable:= Servo_Enable  , 
	bMoveVelocity:= , 
	bHalt:= , 
	bManualMode:= OP10A_MANUAL_SELECTED , 
	fHomePos:= , 
	fOverride:= , 
	fTargetPosition:= OP10A_SRV_RH_BDYANG_CNT.Position, 
	fTargetVelocity:= OP10_SERVO_POS_VEL_LIMIT.OP10A_RH_ROTRY_VELOCITY, 
	fAcc:= , 
	fDec:= ,
	Servo_High_Limit:= OP10_SERVO_POS_VEL_LIMIT.OP10A_RH_ROTRY_POS_LIMIT,																	
	Servo_Low_Limit:=OP10_SERVO_POS_VEL_LIMIT.OP10A_RH_GRPR_NEG_LIMIT, 
	Safe_move_Conditions:= Servo_Safety,
	TORQUE_APPLIED :=  , 
	Axis:= OP10A_RH_ROTARY, 
	bHome:= OP10A_SRV_RH_BDYANG_CNT.Axis_Home_Cmd, 
	bSetPosition:= FESTO_NOT_NEED , 
	bMoveAbsolute:= OP10A_SRV_RH_BDYANG_CNT.ABSmove_Start, 
	bMoveRelative:= NOT_REQ , 
	bMoveTorque:= NOT_REQ , 
	stManualModeAxis:= OP10A_SRV_RH_BDYANG_STUS, 
 	sAxisState=> OP10A_SRV_RH_BDYANG_CNT.Axis_State, 
	bAxis_ready=> , 
	bAxisInPosition=> , 
	bAxisError=> OP10A_SRV_RH_BDYANG_CNT.Axis_Error, 
	bAxisEnabled=> , 
	bAxisHomed=> , 
	bSetPositionDone=> , 
	bHaltDone=> , 
	bSTOPDone=> , 
	bHomeDone=> OP10A_SRV_RH_BDYANG_CNT.Axis_In_Home, 
	bDone=> , 
	bTorqueReached=> , 
	bsafe_to_move=> , 
	baxis_in_home_pos=> , 
	bABS_Pos_done=>OP10A_SRV_RH_BDYANG_CNT.Axis_In_Pos, 
	Actual_position=>,
	Actual_velocity=> , 
	Actual_Torque=> );
	
OP10A_LH_GRIPR(
	bAxis1_Ref_Switch:= , 
	bInit:= OP10_SRV_BLCK_INTZ , 
	bErrorReset:= Servo_Reset, 
	bEnable:= Servo_Enable  , 
	bMoveVelocity:=, 
	bHalt:= , 
	bManualMode:= OP10A_MANUAL_SELECTED , 
	fHomePos:= , 
	fOverride:= , 
	fTargetPosition:= OP10A_SRV_LH_BDYGRP_CNT.Position, 
	fTargetVelocity:= OP10_SERVO_POS_VEL_LIMIT.OP10A_LH_GRPR_VELOCITY, 
	fAcc:= , 
	fDec:= ,
	Servo_High_Limit:= OP10_SERVO_POS_VEL_LIMIT.OP10A_LH_GRPR_POS_LIMIT,																	
	Servo_Low_Limit:=OP10_SERVO_POS_VEL_LIMIT.OP10A_LH_GRPR_NEG_LIMIT, 
	Safe_move_Conditions:= Servo_Safety,
	TORQUE_APPLIED := OP10A_LH_GRP_TORQUE_APPLIED, 
	Axis:= OP10A_LH_GRIPPER, 
	bHome:= OP10A_SRV_LH_BDYGRP_CNT.Axis_Home_Cmd, 
	bSetPosition:= FESTO_NOT_NEED , 
	bMoveAbsolute:= OP10A_SRV_LH_BDYGRP_CNT.ABSmove_Start, 
	bMoveRelative:= NOT_REQ , 
	bMoveTorque:= NOT_REQ , 
	stManualModeAxis:= OP10A_SRV_LH_BDYGRP_STUS, 
 	sAxisState=> OP10A_SRV_LH_BDYGRP_CNT.Axis_State, 
	bAxis_ready=> , 
	bAxisInPosition=> , 
	bAxisError=> OP10A_SRV_LH_BDYGRP_CNT.Axis_Error, 
	bAxisEnabled=> , 
	bAxisHomed=> , 
	bSetPositionDone=> , 
	bHaltDone=> , 
	bSTOPDone=> , 
	bHomeDone=> OP10A_SRV_LH_BDYGRP_CNT.Axis_In_Home, 
	bDone=> , 
	bTorqueReached=> , 
	bsafe_to_move=> , 
	baxis_in_home_pos=> , 
	bABS_Pos_done=> OP10A_SRV_LH_BDYGRP_CNT.Axis_In_Pos, 
	Actual_position=>, 
	Actual_velocity=> , 
	Actual_Torque=> );
	
OP10A_RH_GRIPR(
	bAxis1_Ref_Switch:= , 
	bInit:= OP10_SRV_BLCK_INTZ , 
	bErrorReset:= Servo_Reset, 
	bEnable:= Servo_Enable , 
	bMoveVelocity:= , 
	bHalt:= , 
	bManualMode:= OP10A_MANUAL_SELECTED , 
	fHomePos:= , 
	fOverride:= , 
	fTargetPosition:= OP10A_SRV_RH_BDYGRP_CNT.Position, 
	fTargetVelocity:= OP10_SERVO_POS_VEL_LIMIT.OP10A_RH_GRPR_VELOCITY, 
	fAcc:= , 
	fDec:= ,
	Servo_High_Limit:= OP10_SERVO_POS_VEL_LIMIT.OP10A_RH_GRPR_POS_LIMIT,
    Servo_Low_Limit:=OP10_SERVO_POS_VEL_LIMIT.OP10A_RH_GRPR_NEG_LIMIT,
	Safe_move_Conditions:= Servo_Safety,
	TORQUE_APPLIED := OP10A_RH_GRP_TORQUE_APPLIED, 
	Axis:= OP10A_RH_GRIPPER, 
	bHome:= OP10A_SRV_RH_BDYGRP_CNT.Axis_Home_Cmd, 
	bSetPosition:= FESTO_NOT_NEED , 
	bMoveAbsolute:= OP10A_SRV_RH_BDYGRP_CNT.ABSmove_Start, 
	bMoveRelative:= NOT_REQ , 
	bMoveTorque:= NOT_REQ , 
	stManualModeAxis:= OP10A_SRV_RH_BDYGRP_STUS, 
 	sAxisState=> OP10A_SRV_RH_BDYGRP_CNT.Axis_State, 
	bAxis_ready=> , 
	bAxisInPosition=> , 
	bAxisError=> OP10A_SRV_RH_BDYGRP_CNT.Axis_Error, 
	bAxisEnabled=> , 
	bAxisHomed=> , 
	bSetPositionDone=> , 
	bHaltDone=> , 
	bSTOPDone=> , 
	bHomeDone=> OP10A_SRV_RH_BDYGRP_CNT.Axis_In_Home, 
	bDone=> , 
	bTorqueReached=> , 
	bsafe_to_move=> , 
	baxis_in_home_pos=> , 
	bABS_Pos_done=> OP10A_SRV_RH_BDYGRP_CNT.Axis_In_Pos, 
	Actual_position=>,
	Actual_velocity=> , 
	Actual_Torque=> );

	
OP10A_CONVEYOR(
	bAxis1_Ref_Switch:= , 
	bInit:= OP10_SRV_BLCK_INTZ, 
	bErrorReset:=  Servo_Reset, 
	bEnable:= Servo_Enable , 
	bMoveVelocity:=OP10A_SRV_O_CNVY_CNT.VELmove_Start , 
	bHalt:= , 
	bManualMode:= OP10A_MANUAL_SELECTED,
	fHomePos:= , 
	fOverride:= , 
	fTargetPosition:= OP10A_SRV_O_CNVY_CNT.Position, 
	fTargetVelocity:= OP10A_SRV_O_CNVY_CNT.Velocity, 
	fAcc:= , 
	fDec:= ,
	Safe_move_Conditions:= Servo_Safety, 
	Axis:= OP10A_CONVRY, 
	HME_WRITE_ADD:= 16#5002,	
	bHome:= OP10A_SRV_O_CNVY_CNT.Bsethome, 
	bSetPosition:= OP10A_SRV_O_CNVY_CNT.BsetPos, 
	bMoveAbsolute:= OP10A_SRV_O_CNVY_CNT.ABSmove_Start, 
	bMoveRelative:= OP10A_SRV_O_CNVY_CNT.RELmove_Start , 
	bMoveTorque:= OP10A_SRV_O_CNVY_CNT.Torque_mode_Start, 
	stManualModeAxis:= OP10A_SRV_O_CNVY_STUS , 
	bmove_home:= OP10A_SRV_O_CNVY_CNT.Axis_Home_Cmd, 
	sAxisState=> OP10A_SRV_O_CNVY_CNT.Axis_State, 
	bAxis_ready=> OP10A_SRV_O_CNVY_CNT.Axis_ready,
	bAxisInPosition=> , 
	bAxisError=> OP10A_SRV_O_CNVY_CNT.Axis_Error, 
	bAxisEnabled=> , 
	bAxisHomed=> , 
	bSetPositionDone=> , 
	bHaltDone=> , 
	bSTOPDone=> , 
	bHomeDone=> OP10A_SRV_O_CNVY_CNT.Axis_In_Home, 
	bDone=> , 
	bTorqueReached=> , 
	bsafe_to_move=> , 
	baxis_in_home_pos=> , 
	bABS_Pos_done=> , 
	Actual_position=> OP10A_SRV_O_CNVY_CNT.Actual_Position, 
	Actual_velocity=> OP10A_SRV_O_CNVY_CNT.Actual_Velocity, 
	Actual_Torque=> );
	
	
	
	
	
	
//////////////////////////////////////	OP10B	///////////////////////////////////////////////////////


OP10B_LH_ROTY(
	bAxis1_Ref_Switch:= , 
	bInit:= OP10_SRV_BLCK_INTZ , 
	bErrorReset:= Servo_Reset, 
	bEnable:= Servo_Enable  , 
	bMoveVelocity:= , 
	bHalt:= , 
	bManualMode:= OP10B_MANUAL_SELECTED , 
	fHomePos:= , 
	fOverride:= , 
	fTargetPosition:= OP10B_SRV_LH_BDYANG_CNT.Position, 
	fTargetVelocity:= OP10_SERVO_POS_VEL_LIMIT.OP10B_LH_ROTRY_VELOCITY, 
	fAcc:= , 
	fDec:= ,
	Servo_High_Limit:= OP10_SERVO_POS_VEL_LIMIT.OP10B_LH_ROTRY_POS_LIMIT,
    Servo_Low_Limit:=OP10_SERVO_POS_VEL_LIMIT.OP10B_LH_ROTRY_NEG_LIMIT, 
	Safe_move_Conditions:= Servo_Safety,
	TORQUE_APPLIED := , 
	Axis:= OP10B_LH_ROTARY, 
	bHome:= OP10B_SRV_LH_BDYANG_CNT.Axis_Home_Cmd, 
	bSetPosition:= FESTO_NOT_NEED , 
	bMoveAbsolute:= OP10B_SRV_LH_BDYANG_CNT.ABSmove_Start, 
	bMoveRelative:= NOT_REQ , 
	bMoveTorque:= NOT_REQ , 
	stManualModeAxis:= OP10B_SRV_LH_BDYANG_STUS, 
	sAxisState=> OP10B_SRV_LH_BDYANG_CNT.Axis_State, 
	bAxis_ready=> , 
	bAxisInPosition=> , 
	bAxisError=> OP10B_SRV_LH_BDYANG_CNT.Axis_Error, 
	bAxisEnabled=> , 
	bAxisHomed=> , 
	bSetPositionDone=> , 
	bHaltDone=> , 
	bSTOPDone=> , 
	bHomeDone=>  OP10B_SRV_LH_BDYANG_CNT.Axis_In_Home, 
	bDone=> , 
	bTorqueReached=> , 
	bsafe_to_move=> , 
	baxis_in_home_pos=> , 
	bABS_Pos_done=>OP10B_SRV_LH_BDYANG_CNT.Axis_In_Pos , 
	Actual_position=>,
	Actual_velocity=> , 
	Actual_Torque=> );
	
